LIN {X 0,Y 403.165,Z 557.03,A -85,B 0,C 180,E1 10218.684,E2 10218.684} C_VEL
LIN {X 0,Y 403.207,Z 557.03,A -85,B 0,C 180,E1 10225.722,E2 10225.722} C_VEL
LIN {X 0,Y 403.44,Z 557.03,A -85,B 0,C 180,E1 10233.237,E2 10233.237} C_VEL
LIN {X 0,Y 403.729,Z 557.03,A -85,B 0,C 180,E1 10240.276,E2 10240.276} C_VEL
LIN {X 0,Y 403.994,Z 557.03,A -85,B 0,C 180,E1 10247.007,E2 10247.007} C_VEL
LIN {X 0,Y 404.192,Z 557.03,A -85,B 0,C 180,E1 10253.549,E2 10253.549} C_VEL
LIN {X 0,Y 404.54,Z 557.03,A -85,B 0,C 180,E1 10260,E2 10260} C_VEL
LIN {X 0,Y 404.221,Z 557.03,A -85,B 0,C 180,E1 10266.452,E2 10266.452} C_VEL
LIN {X 0,Y 403.903,Z 557.03,A -85,B 0,C 180,E1 10272.997,E2 10272.997} C_VEL
LIN {X 0,Y 403.588,Z 557.03,A -85,B 0,C 180,E1 10280.305,E2 10280.305} C_VEL
LIN {X 0,Y 403.428,Z 557.03,A -85,B 0,C 180,E1 10286.765,E2 10286.765} C_VEL
LIN {X 0,Y 403.272,Z 557.03,A -85,B 0,C 180,E1 10291.708,E2 10291.708} C_VEL
LIN {X 0,Y 403.118,Z 557.03,A -85,B 0,C 180,E1 10297.934,E2 10297.934} C_VEL
LIN {X 0,Y 403.276,Z 557.65,A -85,B 0,C 180,E1 10303.8,E2 10303.8} C_VEL
LIN {X 0,Y 426.424,Z 601.688,A -85,B 0,C 180,E1 10307.749,E2 10307.749} C_VEL
LIN {X 0,Y 436.03,Z 627.386,A -85,B 0,C 180,E1 10309.651,E2 10309.651} C_VEL
LIN {X 0,Y 431.949,Z 666.261,A -85,B 0,C 180,E1 10311.298,E2 10311.298} C_VEL
LIN {X 0,Y 426.944,Z 703.511,A -85,B 0,C 180,E1 10313.718,E2 10313.718} C_VEL
LIN {X 0,Y 421.04,Z 740.02,A -85,B 0,C 180,E1 10317.052,E2 10317.052} C_VEL
LIN {X 0,Y 415.393,Z 772.458,A -85,B 0,C 180,E1 10321.118,E2 10321.118} C_VEL
LIN {X 0,Y 410.738,Z 800.362,A -85,B 0,C 180,E1 10325.811,E2 10325.811} C_VEL
LIN {X 0,Y 407.625,Z 822.502,A -85,B 0,C 180,E1 10330.852,E2 10330.852} C_VEL
LIN {X 0,Y 406.966,Z 827.151,A -85,B 0,C 180,E1 10332.15,E2 10332.15} C_VEL
LIN {X 0,Y 402.175,Z 834.199,A -85,B 0,C 180,E1 10334.327,E2 10334.327} C_VEL
LIN {X 0,Y 397.666,Z 840.297,A -85,B 0,C 180,E1 10336.6,E2 10336.6} C_VEL
LIN {X 0,Y 397.045,Z 849.258,A -85,B 0,C 180,E1 10341.227,E2 10341.227} C_VEL
LIN {X 0,Y 396.776,Z 854.259,A -85,B 0,C 180,E1 10345.623,E2 10345.623} C_VEL
LIN {X 0,Y 396.836,Z 855.967,A -85,B 0,C 180,E1 10350,E2 10350} C_VEL
LIN {X 0,Y 396.833,Z 853.357,A -85,B 0,C 180,E1 10355.474,E2 10355.474} C_VEL
LIN {X 0,Y 397.276,Z 845.463,A -85,B 0,C 180,E1 10360.986,E2 10360.986} C_VEL
LIN {X 0,Y 398.586,Z 831.788,A -85,B 0,C 180,E1 10366.553,E2 10366.553} C_VEL
LIN {X 0,Y 401.185,Z 812.548,A -85,B 0,C 180,E1 10371.881,E2 10371.881} C_VEL
LIN {X 0,Y 405.349,Z 787.469,A -85,B 0,C 180,E1 10376.93,E2 10376.93} C_VEL
LIN {X 0,Y 410.746,Z 757.402,A -85,B 0,C 180,E1 10381.419,E2 10381.419} C_VEL
LIN {X 0,Y 416.603,Z 724.967,A -85,B 0,C 180,E1 10385.02,E2 10385.02} C_VEL
LIN {X 0,Y 422.428,Z 688.774,A -85,B 0,C 180,E1 10387.958,E2 10387.958} C_VEL
LIN {X 0,Y 427.491,Z 650.452,A -85,B 0,C 180,E1 10390.101,E2 10390.101} C_VEL
LIN {X 0,Y 429.146,Z 626.905,A -85,B 0,C 180,E1 10391.084,E2 10391.084} C_VEL
LIN {X 0,Y 415.014,Z 593.65,A -85,B 0,C 180,E1 10393.806,E2 10393.806} C_VEL
LIN {X 0,Y 397.196,Z 562.149,A -85,B 0,C 180,E1 10396.941,E2 10396.941} C_VEL
LIN {X 0,Y 395.293,Z 557.03,A -85,B 0,C 180,E1 10397.449,E2 10397.449} C_VEL
LIN {X 0,Y 395.232,Z 557.03,A -85,B 0,C 180,E1 10404.929,E2 10404.929} C_VEL
LIN {X 0,Y 395.398,Z 557.03,A -85,B 0,C 180,E1 10411.729,E2 10411.729} C_VEL
LIN {X 0,Y 395.637,Z 557.03,A -85,B 0,C 180,E1 10417.501,E2 10417.501} C_VEL
LIN {X 0,Y 395.771,Z 557.03,A -85,B 0,C 180,E1 10424.468,E2 10424.468} C_VEL
LIN {X 0,Y 396.146,Z 557.03,A -85,B 0,C 180,E1 10431.206,E2 10431.206} C_VEL
LIN {X 0,Y 396.61,Z 557.03,A -85,B 0,C 180,E1 10437.812,E2 10437.812} C_VEL
LIN {X 0,Y 396.445,Z 557.03,A -85,B 0,C 180,E1 10444.38,E2 10444.38} C_VEL
LIN {X 0,Y 396.051,Z 557.03,A -85,B 0,C 180,E1 10451.018,E2 10451.018} C_VEL
LIN {X 0,Y 395.86,Z 557.03,A -85,B 0,C 180,E1 10457.815,E2 10457.815} C_VEL
LIN {X 0,Y 395.54,Z 557.03,A -85,B 0,C 180,E1 10464.899,E2 10464.899} C_VEL
LIN {X 0,Y 395.4,Z 557.03,A -85,B 0,C 180,E1 10469.851,E2 10469.851} C_VEL
LIN {X 0,Y 395.176,Z 557.03,A -85,B 0,C 180,E1 10476.43,E2 10476.43} C_VEL
LIN {X 0,Y 395.189,Z 557.03,A -85,B 0,C 180,E1 10483.595,E2 10483.595} C_VEL
LIN {X 0,Y 395.261,Z 557.03,A -85,B 0,C 180,E1 10487.074,E2 10487.074} C_VEL
LIN {X 0,Y 397.693,Z 562.671,A -85,B 0,C 180,E1 10487.578,E2 10487.578} C_VEL
LIN {X 0,Y 418.659,Z 600.152,A -85,B 0,C 180,E1 10491.241,E2 10491.241} C_VEL
LIN {X 0,Y 428.676,Z 623.291,A -85,B 0,C 180,E1 10493.314,E2 10493.314} C_VEL
LIN {X 0,Y 424.543,Z 659.037,A -85,B 0,C 180,E1 10495.067,E2 10495.067} C_VEL
LIN {X 0,Y 419.009,Z 693.568,A -85,B 0,C 180,E1 10497.653,E2 10497.653} C_VEL
LIN {X 0,Y 412.847,Z 725.198,A -85,B 0,C 180,E1 10501.077,E2 10501.077} C_VEL
LIN {X 0,Y 407.204,Z 751.222,A -85,B 0,C 180,E1 10504.979,E2 10504.979} C_VEL
LIN {X 0,Y 402.464,Z 773.712,A -85,B 0,C 180,E1 10509.636,E2 10509.636} C_VEL
LIN {X 0,Y 399.372,Z 790.725,A -85,B 0,C 180,E1 10514.61,E2 10514.61} C_VEL
LIN {X 0,Y 397.661,Z 803.103,A -85,B 0,C 180,E1 10520.134,E2 10520.134} C_VEL
LIN {X 0,Y 397.016,Z 809.778,A -85,B 0,C 180,E1 10525.625,E2 10525.625} C_VEL
LIN {X 0,Y 396.954,Z 811.42,A -85,B 0,C 180,E1 10530,E2 10530} C_VEL
LIN {X 0,Y 397.126,Z 808.803,A -85,B 0,C 180,E1 10535.469,E2 10535.469} C_VEL
LIN {X 0,Y 397.896,Z 800.917,A -85,B 0,C 180,E1 10540.967,E2 10540.967} C_VEL
LIN {X 0,Y 399.978,Z 787.154,A -85,B 0,C 180,E1 10546.493,E2 10546.493} C_VEL
LIN {X 0,Y 403.828,Z 767.438,A -85,B 0,C 180,E1 10551.73,E2 10551.73} C_VEL
LIN {X 0,Y 408.723,Z 744.251,A -85,B 0,C 180,E1 10556.097,E2 10556.097} C_VEL
LIN {X 0,Y 414.5,Z 716.892,A -85,B 0,C 180,E1 10559.846,E2 10559.846} C_VEL
LIN {X 0,Y 420.536,Z 684.985,A -85,B 0,C 180,E1 10562.993,E2 10562.993} C_VEL
LIN {X 0,Y 425.681,Z 650.957,A -85,B 0,C 180,E1 10565.307,E2 10565.307} C_VEL
LIN {X 0,Y 428.316,Z 621.671,A -85,B 0,C 180,E1 10566.708,E2 10566.708} C_VEL
LIN {X 0,Y 411.761,Z 586.807,A -85,B 0,C 180,E1 10569.882,E2 10569.882} C_VEL
LIN {X 0,Y 395.357,Z 558.405,A -85,B 0,C 180,E1 10572.754,E2 10572.754} C_VEL
LIN {X 0,Y 395.248,Z 557.03,A -85,B 0,C 180,E1 10572.937,E2 10572.937} C_VEL
LIN {X 0,Y 395.242,Z 557.03,A -85,B 0,C 180,E1 10580.008,E2 10580.008} C_VEL
LIN {X 0,Y 395.268,Z 557.03,A -85,B 0,C 180,E1 10587.574,E2 10587.574} C_VEL
LIN {X 0,Y 395.445,Z 557.03,A -85,B 0,C 180,E1 10592.651,E2 10592.651} C_VEL
LIN {X 0,Y 395.802,Z 557.03,A -85,B 0,C 180,E1 10599.864,E2 10599.864} C_VEL
LIN {X 0,Y 396.053,Z 557.03,A -85,B 0,C 180,E1 10606.741,E2 10606.741} C_VEL
LIN {X 0,Y 396.284,Z 557.03,A -85,B 0,C 180,E1 10613.419,E2 10613.419} C_VEL
LIN {X 0,Y 396.638,Z 557.03,A -85,B 0,C 180,E1 10620,E2 10620} C_VEL
LIN {X 0,Y 396.306,Z 557.03,A -85,B 0,C 180,E1 10626.637,E2 10626.637} C_VEL
LIN {X 0,Y 395.957,Z 557.03,A -85,B 0,C 180,E1 10633.263,E2 10633.263} C_VEL
LIN {X 0,Y 395.725,Z 557.03,A -85,B 0,C 180,E1 10640.141,E2 10640.141} C_VEL
LIN {X 0,Y 395.436,Z 557.03,A -85,B 0,C 180,E1 10647.35,E2 10647.35} C_VEL
LIN {X 0,Y 395.287,Z 557.03,A -85,B 0,C 180,E1 10652.579,E2 10652.579} C_VEL
LIN {X 0,Y 395.249,Z 557.03,A -85,B 0,C 180,E1 10659.993,E2 10659.993} C_VEL
LIN {X 0,Y 395.305,Z 557.034,A -85,B 0,C 180,E1 10662.665,E2 10662.665} C_VEL
LIN {X 0,Y 397.735,Z 562.702,A -85,B 0,C 180,E1 10663.162,E2 10663.162} C_VEL
LIN {X 0,Y 417.577,Z 598.711,A -85,B 0,C 180,E1 10666.649,E2 10666.649} C_VEL
LIN {X 0,Y 429.63,Z 629.235,A -85,B 0,C 180,E1 10669.068,E2 10669.068} C_VEL
LIN {X 0,Y 425.163,Z 669.268,A -85,B 0,C 180,E1 10670.836,E2 10670.836} C_VEL
LIN {X 0,Y 419.577,Z 707.742,A -85,B 0,C 180,E1 10673.459,E2 10673.459} C_VEL
LIN {X 0,Y 413.477,Z 742.914,A -85,B 0,C 180,E1 10676.845,E2 10676.845} C_VEL
LIN {X 0,Y 407.709,Z 774.237,A -85,B 0,C 180,E1 10680.937,E2 10680.937} C_VEL
LIN {X 0,Y 403.02,Z 800.884,A -85,B 0,C 180,E1 10685.592,E2 10685.592} C_VEL
LIN {X 0,Y 399.745,Z 823.015,A -85,B 0,C 180,E1 10690.796,E2 10690.796} C_VEL
LIN {X 0,Y 397.756,Z 839.4,A -85,B 0,C 180,E1 10696.238,E2 10696.238} C_VEL
LIN {X 0,Y 397.666,Z 840.297,A -85,B 0,C 180,E1 10696.6,E2 10696.6} C_VEL
LIN {X 0,Y 394.853,Z 844.248,A -85,B 0,C 180,E1 10698.366,E2 10698.366} C_VEL
LIN {X 0,Y 389.243,Z 848.814,A -85,B 0,C 180,E1 10701.079,E2 10701.079} C_VEL
LIN {X 0,Y 389.109,Z 849.256,A -85,B 0,C 180,E1 10701.397,E2 10701.397} C_VEL
LIN {X 0,Y 388.883,Z 853.803,A -85,B 0,C 180,E1 10705.534,E2 10705.534} C_VEL
LIN {X 0,Y 388.961,Z 855.525,A -85,B 0,C 180,E1 10710,E2 10710} C_VEL
LIN {X 0,Y 388.958,Z 852.896,A -85,B 0,C 180,E1 10715.585,E2 10715.585} C_VEL
LIN {X 0,Y 389.415,Z 844.941,A -85,B 0,C 180,E1 10721.21,E2 10721.21} C_VEL
LIN {X 0,Y 390.597,Z 832.802,A -85,B 0,C 180,E1 10726.322,E2 10726.322} C_VEL
LIN {X 0,Y 393.13,Z 814.175,A -85,B 0,C 180,E1 10731.758,E2 10731.758} C_VEL
LIN {X 0,Y 397.32,Z 790.516,A -85,B 0,C 180,E1 10736.792,E2 10736.792} C_VEL
LIN {X 0,Y 402.866,Z 761.455,A -85,B 0,C 180,E1 10741.398,E2 10741.398} C_VEL
LIN {X 0,Y 409.308,Z 727.729,A -85,B 0,C 180,E1 10745.337,E2 10745.337} C_VEL
LIN {X 0,Y 415.569,Z 691.107,A -85,B 0,C 180,E1 10748.421,E2 10748.421} C_VEL
LIN {X 0,Y 420.858,Z 653.779,A -85,B 0,C 180,E1 10750.596,E2 10750.596} C_VEL
LIN {X 0,Y 422.862,Z 629.874,A -85,B 0,C 180,E1 10751.636,E2 10751.636} C_VEL
LIN {X 0,Y 409.373,Z 597.325,A -85,B 0,C 180,E1 10754.401,E2 10754.401} C_VEL
LIN {X 0,Y 389.835,Z 562.756,A -85,B 0,C 180,E1 10758.002,E2 10758.002} C_VEL
LIN {X 0,Y 387.326,Z 557.03,A -85,B 0,C 180,E1 10758.636,E2 10758.636} C_VEL
LIN {X 0,Y 387.322,Z 557.03,A -85,B 0,C 180,E1 10765.175,E2 10765.175} C_VEL
LIN {X 0,Y 387.524,Z 557.03,A -85,B 0,C 180,E1 10772.043,E2 10772.043} C_VEL
LIN {X 0,Y 387.827,Z 557.03,A -85,B 0,C 180,E1 10779.546,E2 10779.546} C_VEL
LIN {X 0,Y 387.914,Z 557.03,A -85,B 0,C 180,E1 10786.457,E2 10786.457} C_VEL
LIN {X 0,Y 388.421,Z 557.03,A -85,B 0,C 180,E1 10793.285,E2 10793.285} C_VEL
LIN {X 0,Y 388.735,Z 557.03,A -85,B 0,C 180,E1 10800,E2 10800} C_VEL
LIN {X 0,Y 388.344,Z 557.03,A -85,B 0,C 180,E1 10806.716,E2 10806.716} C_VEL
LIN {X 0,Y 388.046,Z 557.03,A -85,B 0,C 180,E1 10813.537,E2 10813.537} C_VEL
LIN {X 0,Y 387.809,Z 557.03,A -85,B 0,C 180,E1 10820.569,E2 10820.569} C_VEL
LIN {X 0,Y 387.523,Z 557.03,A -85,B 0,C 180,E1 10827.956,E2 10827.956} C_VEL
LIN {X 0,Y 387.311,Z 557.03,A -85,B 0,C 180,E1 10834.822,E2 10834.822} C_VEL
LIN {X 0,Y 387.177,Z 557.03,A -85,B 0,C 180,E1 10842.012,E2 10842.012} C_VEL
LIN {X 0,Y 387.256,Z 557.03,A -85,B 0,C 180,E1 10845.866,E2 10845.866} C_VEL
LIN {X 0,Y 389.727,Z 562.663,A -85,B 0,C 180,E1 10846.407,E2 10846.407} C_VEL
LIN {X 0,Y 410.465,Z 598.787,A -85,B 0,C 180,E1 10850.187,E2 10850.187} C_VEL
LIN {X 0,Y 422.263,Z 626.321,A -85,B 0,C 180,E1 10852.752,E2 10852.752} C_VEL
LIN {X 0,Y 417.71,Z 662.884,A -85,B 0,C 180,E1 10854.634,E2 10854.634} C_VEL
LIN {X 0,Y 411.761,Z 697.232,A -85,B 0,C 180,E1 10857.345,E2 10857.345} C_VEL
LIN {X 0,Y 405.683,Z 726.809,A -85,B 0,C 180,E1 10860.67,E2 10860.67} C_VEL
LIN {X 0,Y 399.636,Z 753.308,A -85,B 0,C 180,E1 10864.772,E2 10864.772} C_VEL
LIN {X 0,Y 394.76,Z 775.372,A -85,B 0,C 180,E1 10869.514,E2 10869.514} C_VEL
LIN {X 0,Y 391.414,Z 792.87,A -85,B 0,C 180,E1 10874.938,E2 10874.938} C_VEL
LIN {X 0,Y 389.824,Z 803.564,A -85,B 0,C 180,E1 10879.934,E2 10879.934} C_VEL
LIN {X 0,Y 389.162,Z 810.223,A -85,B 0,C 180,E1 10885.537,E2 10885.537} C_VEL
LIN {X 0,Y 389.072,Z 811.863,A -85,B 0,C 180,E1 10890,E2 10890} C_VEL
LIN {X 0,Y 389.245,Z 809.254,A -85,B 0,C 180,E1 10895.58,E2 10895.58} C_VEL
LIN {X 0,Y 390.087,Z 801.385,A -85,B 0,C 180,E1 10901.19,E2 10901.19} C_VEL
LIN {X 0,Y 392.032,Z 789.292,A -85,B 0,C 180,E1 10906.26,E2 10906.26} C_VEL
LIN {X 0,Y 395.574,Z 771.558,A -85,B 0,C 180,E1 10911.322,E2 10911.322} C_VEL
LIN {X 0,Y 400.839,Z 748.189,A -85,B 0,C 180,E1 10916.046,E2 10916.046} C_VEL
LIN {X 0,Y 406.919,Z 720.875,A -85,B 0,C 180,E1 10919.998,E2 10919.998} C_VEL
LIN {X 0,Y 413.186,Z 689.835,A -85,B 0,C 180,E1 10923.225,E2 10923.225} C_VEL
LIN {X 0,Y 418.676,Z 656.143,A -85,B 0,C 180,E1 10925.681,E2 10925.681} C_VEL
LIN {X 0,Y 422.007,Z 624.706,A -85,B 0,C 180,E1 10927.261,E2 10927.261} C_VEL
LIN {X 0,Y 406.748,Z 591.728,A -85,B 0,C 180,E1 10930.396,E2 10930.396} C_VEL
LIN {X 0,Y 387.461,Z 558.663,A -85,B 0,C 180,E1 10933.931,E2 10933.931} C_VEL
LIN {X 0,Y 387.254,Z 557.03,A -85,B 0,C 180,E1 10934.205,E2 10934.205} C_VEL
LIN {X 0,Y 387.263,Z 557.03,A -85,B 0,C 180,E1 10941.436,E2 10941.436} C_VEL
LIN {X 0,Y 387.312,Z 557.03,A -85,B 0,C 180,E1 10946.823,E2 10946.823} C_VEL
LIN {X 0,Y 387.533,Z 557.03,A -85,B 0,C 180,E1 10953.972,E2 10953.972} C_VEL
LIN {X 0,Y 387.839,Z 557.03,A -85,B 0,C 180,E1 10959.538,E2 10959.538} C_VEL
LIN {X 0,Y 388.11,Z 557.03,A -85,B 0,C 180,E1 10966.465,E2 10966.465} C_VEL
LIN {X 0,Y 388.391,Z 557.03,A -85,B 0,C 180,E1 10973.285,E2 10973.285} C_VEL
LIN {X 0,Y 388.743,Z 557.03,A -85,B 0,C 180,E1 10980,E2 10980} C_VEL
LIN {X 0,Y 388.417,Z 557.03,A -85,B 0,C 180,E1 10986.715,E2 10986.715} C_VEL
LIN {X 0,Y 388.028,Z 557.03,A -85,B 0,C 180,E1 10993.539,E2 10993.539} C_VEL
LIN {X 0,Y 387.754,Z 557.03,A -85,B 0,C 180,E1 11000.573,E2 11000.573} C_VEL
LIN {X 0,Y 387.522,Z 557.03,A -85,B 0,C 180,E1 11007.957,E2 11007.957} C_VEL
LIN {X 0,Y 387.285,Z 557.03,A -85,B 0,C 180,E1 11015.9,E2 11015.9} C_VEL
LIN {X 0,Y 387.346,Z 557.03,A -85,B 0,C 180,E1 11021.455,E2 11021.455} C_VEL
LIN {X 0,Y 389.796,Z 562.725,A -85,B 0,C 180,E1 11022.006,E2 11022.006} C_VEL
LIN {X 0,Y 409.799,Z 598.084,A -85,B 0,C 180,E1 11025.683,E2 11025.683} C_VEL
LIN {X 0,Y 423.233,Z 630.882,A -85,B 0,C 180,E1 11028.452,E2 11028.452} C_VEL
LIN {X 0,Y 418.376,Z 672.307,A -85,B 0,C 180,E1 11030.371,E2 11030.371} C_VEL
LIN {X 0,Y 412.773,Z 708.514,A -85,B 0,C 180,E1 11032.921,E2 11032.921} C_VEL
LIN {X 0,Y 406.381,Z 743.419,A -85,B 0,C 180,E1 11036.354,E2 11036.354} C_VEL
LIN {X 0,Y 400.543,Z 773.668,A -85,B 0,C 180,E1 11040.382,E2 11040.382} C_VEL
LIN {X 0,Y 395.53,Z 800.233,A -85,B 0,C 180,E1 11045.098,E2 11045.098} C_VEL
LIN {X 0,Y 392.058,Z 822.04,A -85,B 0,C 180,E1 11050.321,E2 11050.321} C_VEL
LIN {X 0,Y 389.986,Z 838.416,A -85,B 0,C 180,E1 11055.79,E2 11055.79} C_VEL
LIN {X 0,Y 389.109,Z 849.256,A -85,B 0,C 180,E1 11061.397,E2 11061.397} C_VEL
LIN {X 0,Y 387.723,Z 850.914,A -85,B 0,C 180,E1 11062.645,E2 11062.645} C_VEL
LIN {X 0,Y 380.923,Z 853.959,A -85,B 0,C 180,E1 11066.339,E2 11066.339} C_VEL
LIN {X 0,Y 380.915,Z 853.897,A -85,B 0,C 180,E1 11066.421,E2 11066.421} C_VEL
LIN {X 0,Y 381.072,Z 855.082,A -85,B 0,C 180,E1 11070,E2 11070} C_VEL
LIN {X 0,Y 380.996,Z 853.345,A -85,B 0,C 180,E1 11074.559,E2 11074.559} C_VEL
LIN {X 0,Y 381.423,Z 846.471,A -85,B 0,C 180,E1 11080.29,E2 11080.29} C_VEL
LIN {X 0,Y 382.457,Z 835.419,A -85,B 0,C 180,E1 11085.499,E2 11085.499} C_VEL
LIN {X 0,Y 385.001,Z 817.102,A -85,B 0,C 180,E1 11091.31,E2 11091.31} C_VEL
LIN {X 0,Y 389.227,Z 793.518,A -85,B 0,C 180,E1 11096.653,E2 11096.653} C_VEL
LIN {X 0,Y 394.728,Z 766.59,A -85,B 0,C 180,E1 11101.186,E2 11101.186} C_VEL
LIN {X 0,Y 401.037,Z 735.014,A -85,B 0,C 180,E1 11105.172,E2 11105.172} C_VEL
LIN {X 0,Y 407.747,Z 699.7,A -85,B 0,C 180,E1 11108.414,E2 11108.414} C_VEL
LIN {X 0,Y 413.272,Z 664.179,A -85,B 0,C 180,E1 11110.736,E2 11110.736} C_VEL
LIN {X 0,Y 416.352,Z 632.035,A -85,B 0,C 180,E1 11112.272,E2 11112.272} C_VEL
LIN {X 0,Y 403.663,Z 600.934,A -85,B 0,C 180,E1 11115.029,E2 11115.029} C_VEL
LIN {X 0,Y 385.101,Z 568.091,A -85,B 0,C 180,E1 11118.578,E2 11118.578} C_VEL
LIN {X 0,Y 379.519,Z 558.27,A -85,B 0,C 180,E1 11119.75,E2 11119.75} C_VEL
LIN {X 0,Y 379.451,Z 557.03,A -85,B 0,C 180,E1 11119.859,E2 11119.859} C_VEL
LIN {X 0,Y 379.436,Z 557.03,A -85,B 0,C 180,E1 11126.926,E2 11126.926} C_VEL
LIN {X 0,Y 379.643,Z 557.03,A -85,B 0,C 180,E1 11133.981,E2 11133.981} C_VEL
LIN {X 0,Y 379.912,Z 557.03,A -85,B 0,C 180,E1 11141.409,E2 11141.409} C_VEL
LIN {X 0,Y 380.062,Z 557.03,A -85,B 0,C 180,E1 11148.511,E2 11148.511} C_VEL
LIN {X 0,Y 380.523,Z 557.03,A -85,B 0,C 180,E1 11155.436,E2 11155.436} C_VEL
LIN {X 0,Y 380.834,Z 557.03,A -85,B 0,C 180,E1 11160,E2 11160} C_VEL
LIN {X 0,Y 380.433,Z 557.03,A -85,B 0,C 180,E1 11166.856,E2 11166.856} C_VEL
LIN {X 0,Y 380.103,Z 557.03,A -85,B 0,C 180,E1 11173.826,E2 11173.826} C_VEL
LIN {X 0,Y 379.831,Z 557.03,A -85,B 0,C 180,E1 11181.021,E2 11181.021} C_VEL
LIN {X 0,Y 379.527,Z 557.03,A -85,B 0,C 180,E1 11188.639,E2 11188.639} C_VEL
LIN {X 0,Y 379.375,Z 557.03,A -85,B 0,C 180,E1 11193.965,E2 11193.965} C_VEL
LIN {X 0,Y 379.212,Z 557.03,A -85,B 0,C 180,E1 11200.659,E2 11200.659} C_VEL
LIN {X 0,Y 379.31,Z 557.559,A -85,B 0,C 180,E1 11204.628,E2 11204.628} C_VEL
LIN {X 0,Y 381.988,Z 562.965,A -85,B 0,C 180,E1 11205.205,E2 11205.205} C_VEL
LIN {X 0,Y 402.845,Z 598.459,A -85,B 0,C 180,E1 11209.186,E2 11209.186} C_VEL
LIN {X 0,Y 415.904,Z 629.213,A -85,B 0,C 180,E1 11212.167,E2 11212.167} C_VEL
LIN {X 0,Y 410.844,Z 666.49,A -85,B 0,C 180,E1 11214.186,E2 11214.186} C_VEL
LIN {X 0,Y 404.765,Z 699.746,A -85,B 0,C 180,E1 11216.927,E2 11216.927} C_VEL
LIN {X 0,Y 398.286,Z 729.434,A -85,B 0,C 180,E1 11220.384,E2 11220.384} C_VEL
LIN {X 0,Y 392.086,Z 755.387,A -85,B 0,C 180,E1 11224.558,E2 11224.558} C_VEL
LIN {X 0,Y 387.036,Z 776.93,A -85,B 0,C 180,E1 11229.385,E2 11229.385} C_VEL
LIN {X 0,Y 383.753,Z 793.018,A -85,B 0,C 180,E1 11234.498,E2 11234.498} C_VEL
LIN {X 0,Y 382.004,Z 804.022,A -85,B 0,C 180,E1 11239.726,E2 11239.726} C_VEL
LIN {X 0,Y 381.28,Z 810.669,A -85,B 0,C 180,E1 11245.444,E2 11245.444} C_VEL
LIN {X 0,Y 381.184,Z 812.305,A -85,B 0,C 180,E1 11250,E2 11250} C_VEL
LIN {X 0,Y 381.389,Z 809.703,A -85,B 0,C 180,E1 11255.695,E2 11255.695} C_VEL
LIN {X 0,Y 382.278,Z 801.851,A -85,B 0,C 180,E1 11261.421,E2 11261.421} C_VEL
LIN {X 0,Y 384.361,Z 789.777,A -85,B 0,C 180,E1 11266.594,E2 11266.594} C_VEL
LIN {X 0,Y 388.17,Z 772.065,A -85,B 0,C 180,E1 11271.749,E2 11271.749} C_VEL
LIN {X 0,Y 393.691,Z 748.737,A -85,B 0,C 180,E1 11276.556,E2 11276.556} C_VEL
LIN {X 0,Y 400.327,Z 720.368,A -85,B 0,C 180,E1 11280.702,E2 11280.702} C_VEL
LIN {X 0,Y 406.818,Z 689.418,A -85,B 0,C 180,E1 11283.935,E2 11283.935} C_VEL
LIN {X 0,Y 412.439,Z 656.42,A -85,B 0,C 180,E1 11286.352,E2 11286.352} C_VEL
LIN {X 0,Y 415.534,Z 627.287,A -85,B 0,C 180,E1 11287.877,E2 11287.877} C_VEL
LIN {X 0,Y 400.346,Z 593.876,A -85,B 0,C 180,E1 11291.19,E2 11291.19} C_VEL
LIN {X 0,Y 381.136,Z 562.063,A -85,B 0,C 180,E1 11294.847,E2 11294.847} C_VEL
LIN {X 0,Y 379.333,Z 557.03,A -85,B 0,C 180,E1 11295.304,E2 11295.304} C_VEL
LIN {X 0,Y 379.252,Z 557.03,A -85,B 0,C 180,E1 11300.305,E2 11300.305} C_VEL
LIN {X 0,Y 379.427,Z 557.03,A -85,B 0,C 180,E1 11306.926,E2 11306.926} C_VEL
LIN {X 0,Y 379.649,Z 557.03,A -85,B 0,C 180,E1 11313.983,E2 11313.983} C_VEL
LIN {X 0,Y 380.001,Z 557.03,A -85,B 0,C 180,E1 11321.415,E2 11321.415} C_VEL
LIN {X 0,Y 380.271,Z 557.03,A -85,B 0,C 180,E1 11328.518,E2 11328.518} C_VEL
LIN {X 0,Y 380.618,Z 557.03,A -85,B 0,C 180,E1 11335.438,E2 11335.438} C_VEL
LIN {X 0,Y 380.795,Z 557.03,A -85,B 0,C 180,E1 11342.279,E2 11342.279} C_VEL
LIN {X 0,Y 380.311,Z 557.03,A -85,B 0,C 180,E1 11349.163,E2 11349.163} C_VEL
LIN {X 0,Y 379.967,Z 557.03,A -85,B 0,C 180,E1 11356.196,E2 11356.196} C_VEL
LIN {X 0,Y 379.716,Z 557.03,A -85,B 0,C 180,E1 11363.498,E2 11363.498} C_VEL
LIN {X 0,Y 379.415,Z 557.03,A -85,B 0,C 180,E1 11371.247,E2 11371.247} C_VEL
LIN {X 0,Y 379.283,Z 557.03,A -85,B 0,C 180,E1 11377.025,E2 11377.025} C_VEL
LIN {X 0,Y 379.431,Z 557.03,A -85,B 0,C 180,E1 11380.203,E2 11380.203} C_VEL
LIN {X 0,Y 381.795,Z 562.637,A -85,B 0,C 180,E1 11380.761,E2 11380.761} C_VEL
LIN {X 0,Y 401.064,Z 595.734,A -85,B 0,C 180,E1 11384.483,E2 11384.483} C_VEL
LIN {X 0,Y 414.31,Z 626.287,A -85,B 0,C 180,E1 11387.245,E2 11387.245} C_VEL
LIN {X 0,Y 416.724,Z 634.752,A -85,B 0,C 180,E1 11387.912,E2 11387.912} C_VEL
LIN {X 0,Y 411.832,Z 673.531,A -85,B 0,C 180,E1 11389.785,E2 11389.785} C_VEL
LIN {X 0,Y 405.961,Z 709.471,A -85,B 0,C 180,E1 11392.377,E2 11392.377} C_VEL
LIN {X 0,Y 399.361,Z 743.852,A -85,B 0,C 180,E1 11395.836,E2 11395.836} C_VEL
LIN {X 0,Y 393.176,Z 774.118,A -85,B 0,C 180,E1 11399.96,E2 11399.96} C_VEL
LIN {X 0,Y 387.84,Z 801.02,A -85,B 0,C 180,E1 11404.879,E2 11404.879} C_VEL
LIN {X 0,Y 384.158,Z 822.955,A -85,B 0,C 180,E1 11410.337,E2 11410.337} C_VEL
LIN {X 0,Y 381.967,Z 839.667,A -85,B 0,C 180,E1 11416.242,E2 11416.242} C_VEL
LIN {X 0,Y 381.172,Z 849.92,A -85,B 0,C 180,E1 11422.009,E2 11422.009} C_VEL
LIN {X 0,Y 380.915,Z 853.897,A -85,B 0,C 180,E1 11426.421,E2 11426.421} C_VEL
LIN {X 0,Y 378.401,Z 854.68,A -85,B 0,C 180,E1 11428.361,E2 11428.361} C_VEL
LIN {X 0,Y 373.165,Z 854.446,A -85,B 0,C 180,E1 11431.291,E2 11431.291} C_VEL
LIN {X 0,Y 373.082,Z 854.32,A -85,B 0,C 180,E1 11431.63,E2 11431.63} C_VEL
LIN {X 0,Y 373.224,Z 850.761,A -85,B 0,C 180,E1 11436.991,E2 11436.991} C_VEL
LIN {X 0,Y 373.918,Z 841.866,A -85,B 0,C 180,E1 11442.741,E2 11442.741} C_VEL
LIN {X 0,Y 375.548,Z 828.32,A -85,B 0,C 180,E1 11448.207,E2 11448.207} C_VEL
LIN {X 0,Y 378.856,Z 808.257,A -85,B 0,C 180,E1 11453.869,E2 11453.869} C_VEL
LIN {X 0,Y 383.938,Z 783.144,A -85,B 0,C 180,E1 11459.036,E2 11459.036} C_VEL
LIN {X 0,Y 390.335,Z 753.565,A -85,B 0,C 180,E1 11463.548,E2 11463.548} C_VEL
LIN {X 0,Y 397.159,Z 720.956,A -85,B 0,C 180,E1 11467.224,E2 11467.224} C_VEL
LIN {X 0,Y 403.984,Z 683.397,A -85,B 0,C 180,E1 11470.278,E2 11470.278} C_VEL
LIN {X 0,Y 409.731,Z 643.204,A -85,B 0,C 180,E1 11472.452,E2 11472.452} C_VEL
LIN {X 0,Y 409.991,Z 634.595,A -85,B 0,C 180,E1 11472.881,E2 11472.881} C_VEL
LIN {X 0,Y 398.341,Z 605.249,A -85,B 0,C 180,E1 11475.608,E2 11475.608} C_VEL
LIN {X 0,Y 380.757,Z 573.73,A -85,B 0,C 180,E1 11479.105,E2 11479.105} C_VEL
LIN {X 0,Y 371.492,Z 558.119,A -85,B 0,C 180,E1 11481.121,E2 11481.121} C_VEL
LIN {X 0,Y 371.41,Z 557.03,A -85,B 0,C 180,E1 11481.204,E2 11481.204} C_VEL
LIN {X 0,Y 371.509,Z 557.03,A -85,B 0,C 180,E1 11488.853,E2 11488.853} C_VEL
LIN {X 0,Y 371.743,Z 557.03,A -85,B 0,C 180,E1 11495.967,E2 11495.967} C_VEL
LIN {X 0,Y 371.95,Z 557.03,A -85,B 0,C 180,E1 11500.996,E2 11500.996} C_VEL
LIN {X 0,Y 372.122,Z 557.03,A -85,B 0,C 180,E1 11508.263,E2 11508.263} C_VEL
LIN {X 0,Y 372.613,Z 557.03,A -85,B 0,C 180,E1 11515.339,E2 11515.339} C_VEL
LIN {X 0,Y 372.932,Z 557.03,A -85,B 0,C 180,E1 11520,E2 11520} C_VEL
LIN {X 0,Y 372.507,Z 557.03,A -85,B 0,C 180,E1 11527.003,E2 11527.003} C_VEL
LIN {X 0,Y 372.16,Z 557.03,A -85,B 0,C 180,E1 11534.127,E2 11534.127} C_VEL
LIN {X 0,Y 371.857,Z 557.03,A -85,B 0,C 180,E1 11541.494,E2 11541.494} C_VEL
LIN {X 0,Y 371.642,Z 557.03,A -85,B 0,C 180,E1 11546.622,E2 11546.622} C_VEL
LIN {X 0,Y 371.489,Z 557.03,A -85,B 0,C 180,E1 11551.991,E2 11551.991} C_VEL
LIN {X 0,Y 371.271,Z 557.03,A -85,B 0,C 180,E1 11559.21,E2 11559.21} C_VEL
LIN {X 0,Y 371.304,Z 557.03,A -85,B 0,C 180,E1 11563.217,E2 11563.217} C_VEL
LIN {X 0,Y 373.599,Z 562.571,A -85,B 0,C 180,E1 11563.793,E2 11563.793} C_VEL
LIN {X 0,Y 392.02,Z 592.498,A -85,B 0,C 180,E1 11567.498,E2 11567.498} C_VEL
LIN {X 0,Y 406.924,Z 624.183,A -85,B 0,C 180,E1 11570.818,E2 11570.818} C_VEL
LIN {X 0,Y 409.369,Z 633.438,A -85,B 0,C 180,E1 11571.63,E2 11571.63} C_VEL
LIN {X 0,Y 404.25,Z 668.689,A -85,B 0,C 180,E1 11573.634,E2 11573.634} C_VEL
LIN {X 0,Y 397.989,Z 701.283,A -85,B 0,C 180,E1 11576.396,E2 11576.396} C_VEL
LIN {X 0,Y 391.424,Z 730.008,A -85,B 0,C 180,E1 11579.811,E2 11579.811} C_VEL
LIN {X 0,Y 384.891,Z 755.918,A -85,B 0,C 180,E1 11584.047,E2 11584.047} C_VEL
LIN {X 0,Y 379.568,Z 777.42,A -85,B 0,C 180,E1 11588.961,E2 11588.961} C_VEL
LIN {X 0,Y 376.065,Z 793.516,A -85,B 0,C 180,E1 11594.184,E2 11594.184} C_VEL
LIN {X 0,Y 374.185,Z 804.478,A -85,B 0,C 180,E1 11599.509,E2 11599.509} C_VEL
LIN {X 0,Y 373.399,Z 811.115,A -85,B 0,C 180,E1 11605.348,E2 11605.348} C_VEL
LIN {X 0,Y 373.303,Z 812.748,A -85,B 0,C 180,E1 11610,E2 11610} C_VEL
LIN {X 0,Y 373.53,Z 810.154,A -85,B 0,C 180,E1 11615.812,E2 11615.812} C_VEL
LIN {X 0,Y 374.49,Z 802.313,A -85,B 0,C 180,E1 11621.662,E2 11621.662} C_VEL
LIN {X 0,Y 376.708,Z 790.259,A -85,B 0,C 180,E1 11626.941,E2 11626.941} C_VEL
LIN {X 0,Y 380.762,Z 772.568,A -85,B 0,C 180,E1 11632.194,E2 11632.194} C_VEL
LIN {X 0,Y 386.575,Z 749.274,A -85,B 0,C 180,E1 11637.084,E2 11637.084} C_VEL
LIN {X 0,Y 393.526,Z 720.974,A -85,B 0,C 180,E1 11641.291,E2 11641.291} C_VEL
LIN {X 0,Y 400.303,Z 690.115,A -85,B 0,C 180,E1 11644.564,E2 11644.564} C_VEL
LIN {X 0,Y 406.086,Z 657.703,A -85,B 0,C 180,E1 11646.982,E2 11646.982} C_VEL
LIN {X 0,Y 409.199,Z 630.078,A -85,B 0,C 180,E1 11648.49,E2 11648.49} C_VEL
LIN {X 0,Y 394.226,Z 596.613,A -85,B 0,C 180,E1 11651.962,E2 11651.962} C_VEL
LIN {X 0,Y 374.022,Z 562.946,A -85,B 0,C 180,E1 11656.012,E2 11656.012} C_VEL
LIN {X 0,Y 371.47,Z 558.414,A -85,B 0,C 180,E1 11656.58,E2 11656.58} C_VEL
LIN {X 0,Y 371.358,Z 557.03,A -85,B 0,C 180,E1 11656.708,E2 11656.708} C_VEL
LIN {X 0,Y 371.29,Z 557.03,A -85,B 0,C 180,E1 11662.293,E2 11662.293} C_VEL
LIN {X 0,Y 371.504,Z 557.03,A -85,B 0,C 180,E1 11668.853,E2 11668.853} C_VEL
LIN {X 0,Y 371.739,Z 557.03,A -85,B 0,C 180,E1 11675.968,E2 11675.968} C_VEL
LIN {X 0,Y 372.184,Z 557.03,A -85,B 0,C 180,E1 11683.457,E2 11683.457} C_VEL
LIN {X 0,Y 372.421,Z 557.03,A -85,B 0,C 180,E1 11690.642,E2 11690.642} C_VEL
LIN {X 0,Y 372.836,Z 557.03,A -85,B 0,C 180,E1 11697.673,E2 11697.673} C_VEL
LIN {X 0,Y 372.879,Z 557.03,A -85,B 0,C 180,E1 11702.327,E2 11702.327} C_VEL
LIN {X 0,Y 372.372,Z 557.03,A -85,B 0,C 180,E1 11709.36,E2 11709.36} C_VEL
LIN {X 0,Y 372.055,Z 557.03,A -85,B 0,C 180,E1 11716.55,E2 11716.55} C_VEL
LIN {X 0,Y 371.738,Z 557.03,A -85,B 0,C 180,E1 11724.033,E2 11724.033} C_VEL
LIN {X 0,Y 371.486,Z 557.03,A -85,B 0,C 180,E1 11731.992,E2 11731.992} C_VEL
LIN {X 0,Y 371.394,Z 557.03,A -85,B 0,C 180,E1 11738.845,E2 11738.845} C_VEL
LIN {X 0,Y 373.811,Z 562.605,A -85,B 0,C 180,E1 11739.436,E2 11739.436} C_VEL
LIN {X 0,Y 393.198,Z 595.069,A -85,B 0,C 180,E1 11743.379,E2 11743.379} C_VEL
LIN {X 0,Y 406.902,Z 625.475,A -85,B 0,C 180,E1 11746.32,E2 11746.32} C_VEL
LIN {X 0,Y 410.295,Z 637.739,A -85,B 0,C 180,E1 11747.329,E2 11747.329} C_VEL
LIN {X 0,Y 405.186,Z 675.863,A -85,B 0,C 180,E1 11749.251,E2 11749.251} C_VEL
LIN {X 0,Y 399.081,Z 711.121,A -85,B 0,C 180,E1 11751.877,E2 11751.877} C_VEL
LIN {X 0,Y 392.367,Z 744.375,A -85,B 0,C 180,E1 11755.309,E2 11755.309} C_VEL
LIN {X 0,Y 386.069,Z 773.5,A -85,B 0,C 180,E1 11759.348,E2 11759.348} C_VEL
LIN {X 0,Y 380.698,Z 799.054,A -85,B 0,C 180,E1 11764.058,E2 11764.058} C_VEL
LIN {X 0,Y 376.759,Z 820.663,A -85,B 0,C 180,E1 11769.413,E2 11769.413} C_VEL
LIN {X 0,Y 374.504,Z 836.32,A -85,B 0,C 180,E1 11774.765,E2 11774.765} C_VEL
LIN {X 0,Y 373.428,Z 847.778,A -85,B 0,C 180,E1 11780.667,E2 11780.667} C_VEL
LIN {X 0,Y 373.033,Z 853.486,A -85,B 0,C 180,E1 11786.424,E2 11786.424} C_VEL
LIN {X 0,Y 373.082,Z 854.32,A -85,B 0,C 180,E1 11791.63,E2 11791.63} C_VEL
LIN {X 0,Y 370.563,Z 853.472,A -85,B 0,C 180,E1 11793.61,E2 11793.61} C_VEL
LIN {X 0,Y 365.361,Z 850.91,A -85,B 0,C 180,E1 11796.579,E2 11796.579} C_VEL
LIN {X 0,Y 365.315,Z 850.519,A -85,B 0,C 180,E1 11796.921,E2 11796.921} C_VEL
LIN {X 0,Y 366.073,Z 841.58,A -85,B 0,C 180,E1 11802.918,E2 11802.918} C_VEL
LIN {X 0,Y 367.932,Z 827.074,A -85,B 0,C 180,E1 11808.845,E2 11808.845} C_VEL
LIN {X 0,Y 371.369,Z 807.71,A -85,B 0,C 180,E1 11814.381,E2 11814.381} C_VEL
LIN {X 0,Y 376.691,Z 782.944,A -85,B 0,C 180,E1 11819.574,E2 11819.574} C_VEL
LIN {X 0,Y 383.397,Z 753.582,A -85,B 0,C 180,E1 11824.137,E2 11824.137} C_VEL
LIN {X 0,Y 390.39,Z 721.754,A -85,B 0,C 180,E1 11827.798,E2 11827.798} C_VEL
LIN {X 0,Y 397.137,Z 686.433,A -85,B 0,C 180,E1 11830.759,E2 11830.759} C_VEL
LIN {X 0,Y 403.106,Z 647.847,A -85,B 0,C 180,E1 11832.964,E2 11832.964} C_VEL
LIN {X 0,Y 403.708,Z 637.185,A -85,B 0,C 180,E1 11833.5,E2 11833.5} C_VEL
LIN {X 0,Y 392.192,Z 607.731,A -85,B 0,C 180,E1 11836.368,E2 11836.368} C_VEL
LIN {X 0,Y 373.793,Z 574.786,A -85,B 0,C 180,E1 11840.223,E2 11840.223} C_VEL
LIN {X 0,Y 363.494,Z 558.064,A -85,B 0,C 180,E1 11842.586,E2 11842.586} C_VEL
LIN {X 0,Y 363.424,Z 557.03,A -85,B 0,C 180,E1 11842.746,E2 11842.746} C_VEL
LIN {X 0,Y 363.615,Z 557.03,A -85,B 0,C 180,E1 11850.024,E2 11850.024} C_VEL
LIN {X 0,Y 363.878,Z 557.03,A -85,B 0,C 180,E1 11858.009,E2 11858.009} C_VEL
LIN {X 0,Y 364.108,Z 557.03,A -85,B 0,C 180,E1 11865.553,E2 11865.553} C_VEL
LIN {X 0,Y 364.662,Z 557.03,A -85,B 0,C 180,E1 11872.845,E2 11872.845} C_VEL
LIN {X 0,Y 365.03,Z 557.03,A -85,B 0,C 180,E1 11880,E2 11880} C_VEL
LIN {X 0,Y 364.585,Z 557.03,A -85,B 0,C 180,E1 11887.156,E2 11887.156} C_VEL
LIN {X 0,Y 364.216,Z 557.03,A -85,B 0,C 180,E1 11894.442,E2 11894.442} C_VEL
LIN {X 0,Y 363.876,Z 557.03,A -85,B 0,C 180,E1 11901.99,E2 11901.99} C_VEL
LIN {X 0,Y 363.614,Z 557.03,A -85,B 0,C 180,E1 11909.975,E2 11909.975} C_VEL
LIN {X 0,Y 363.373,Z 557.03,A -85,B 0,C 180,E1 11917.658,E2 11917.658} C_VEL
LIN {X 0,Y 363.406,Z 557.521,A -85,B 0,C 180,E1 11921.801,E2 11921.801} C_VEL
LIN {X 0,Y 365.947,Z 562.812,A -85,B 0,C 180,E1 11922.431,E2 11922.431} C_VEL
LIN {X 0,Y 385.714,Z 594.655,A -85,B 0,C 180,E1 11926.625,E2 11926.625} C_VEL
LIN {X 0,Y 400.188,Z 625.792,A -85,B 0,C 180,E1 11930.043,E2 11930.043} C_VEL
LIN {X 0,Y 403.16,Z 635.392,A -85,B 0,C 180,E1 11930.984,E2 11930.984} C_VEL
LIN {X 0,Y 397.688,Z 671.012,A -85,B 0,C 180,E1 11933.076,E2 11933.076} C_VEL
LIN {X 0,Y 390.819,Z 704.673,A -85,B 0,C 180,E1 11936.033,E2 11936.033} C_VEL
LIN {X 0,Y 383.311,Z 735.398,A -85,B 0,C 180,E1 11939.916,E2 11939.916} C_VEL
LIN {X 0,Y 376.535,Z 760.836,A -85,B 0,C 180,E1 11944.422,E2 11944.422} C_VEL
LIN {X 0,Y 371.327,Z 780.87,A -85,B 0,C 180,E1 11949.365,E2 11949.365} C_VEL
LIN {X 0,Y 367.858,Z 796.854,A -85,B 0,C 180,E1 11955.032,E2 11955.032} C_VEL
LIN {X 0,Y 366.181,Z 806.738,A -85,B 0,C 180,E1 11960.48,E2 11960.48} C_VEL
LIN {X 0,Y 365.52,Z 811.56,A -85,B 0,C 180,E1 11965.248,E2 11965.248} C_VEL
LIN {X 0,Y 365.415,Z 813.19,A -85,B 0,C 180,E1 11970,E2 11970} C_VEL
LIN {X 0,Y 365.535,Z 811.492,A -85,B 0,C 180,E1 11974.751,E2 11974.751} C_VEL
LIN {X 0,Y 366.403,Z 804.789,A -85,B 0,C 180,E1 11980.716,E2 11980.716} C_VEL
LIN {X 0,Y 368.733,Z 792.387,A -85,B 0,C 180,E1 11986.703,E2 11986.703} C_VEL
LIN {X 0,Y 373.076,Z 774.218,A -85,B 0,C 180,E1 11992.362,E2 11992.362} C_VEL
LIN {X 0,Y 379.069,Z 751.346,A -85,B 0,C 180,E1 11997.343,E2 11997.343} C_VEL
LIN {X 0,Y 386.264,Z 723.812,A -85,B 0,C 180,E1 12001.618,E2 12001.618} C_VEL
LIN {X 0,Y 393.532,Z 692.309,A -85,B 0,C 180,E1 12005.078,E2 12005.078} C_VEL
LIN {X 0,Y 399.656,Z 659.701,A -85,B 0,C 180,E1 12007.587,E2 12007.587} C_VEL
LIN {X 0,Y 402.952,Z 633.102,A -85,B 0,C 180,E1 12009.086,E2 12009.086} C_VEL
LIN {X 0,Y 388.682,Z 600.276,A -85,B 0,C 180,E1 12012.626,E2 12012.626} C_VEL
LIN {X 0,Y 369.853,Z 568.768,A -85,B 0,C 180,E1 12016.584,E2 12016.584} C_VEL
LIN {X 0,Y 363.577,Z 558.452,A -85,B 0,C 180,E1 12018.023,E2 12018.023} C_VEL
LIN {X 0,Y 363.434,Z 557.03,A -85,B 0,C 180,E1 12018.203,E2 12018.203} C_VEL
LIN {X 0,Y 363.385,Z 557.03,A -85,B 0,C 180,E1 12024.32,E2 12024.32} C_VEL
LIN {X 0,Y 363.662,Z 557.03,A -85,B 0,C 180,E1 12030.962,E2 12030.962} C_VEL
LIN {X 0,Y 363.882,Z 557.03,A -85,B 0,C 180,E1 12038.01,E2 12038.01} C_VEL
LIN {X 0,Y 364.305,Z 557.03,A -85,B 0,C 180,E1 12045.562,E2 12045.562} C_VEL
LIN {X 0,Y 364.639,Z 557.03,A -85,B 0,C 180,E1 12052.845,E2 12052.845} C_VEL
LIN {X 0,Y 365.038,Z 557.03,A -85,B 0,C 180,E1 12060,E2 12060} C_VEL
LIN {X 0,Y 364.665,Z 557.03,A -85,B 0,C 180,E1 12067.155,E2 12067.155} C_VEL
LIN {X 0,Y 364.186,Z 557.03,A -85,B 0,C 180,E1 12074.444,E2 12074.444} C_VEL
LIN {X 0,Y 363.85,Z 557.03,A -85,B 0,C 180,E1 12081.993,E2 12081.993} C_VEL
LIN {X 0,Y 363.611,Z 557.03,A -85,B 0,C 180,E1 12089.976,E2 12089.976} C_VEL
LIN {X 0,Y 363.456,Z 557.742,A -85,B 0,C 180,E1 12097.419,E2 12097.419} C_VEL
LIN {X 0,Y 366.283,Z 563.05,A -85,B 0,C 180,E1 12098.114,E2 12098.114} C_VEL
LIN {X 0,Y 386.389,Z 596.357,A -85,B 0,C 180,E1 12102.428,E2 12102.428} C_VEL
LIN {X 0,Y 400.282,Z 626.878,A -85,B 0,C 180,E1 12105.553,E2 12105.553} C_VEL
LIN {X 0,Y 403.952,Z 640.514,A -85,B 0,C 180,E1 12106.72,E2 12106.72} C_VEL
LIN {X 0,Y 398.374,Z 679.291,A -85,B 0,C 180,E1 12108.765,E2 12108.765} C_VEL
LIN {X 0,Y 391.327,Z 717.197,A -85,B 0,C 180,E1 12111.754,E2 12111.754} C_VEL
LIN {X 0,Y 383.857,Z 751.557,A -85,B 0,C 180,E1 12115.596,E2 12115.596} C_VEL
LIN {X 0,Y 377.01,Z 781.692,A -85,B 0,C 180,E1 12120.208,E2 12120.208} C_VEL
LIN {X 0,Y 371.594,Z 806.443,A -85,B 0,C 180,E1 12125.315,E2 12125.315} C_VEL
LIN {X 0,Y 367.987,Z 826.987,A -85,B 0,C 180,E1 12131.13,E2 12131.13} C_VEL
LIN {X 0,Y 366.011,Z 841.63,A -85,B 0,C 180,E1 12137.107,E2 12137.107} C_VEL
LIN {X 0,Y 365.345,Z 850.297,A -85,B 0,C 180,E1 12142.859,E2 12142.859} C_VEL
LIN {X 0,Y 365.207,Z 853.735,A -85,B 0,C 180,E1 12147.624,E2 12147.624} C_VEL
LIN {X 0,Y 365.228,Z 853.737,A -85,B 0,C 180,E1 12152.376,E2 12152.376} C_VEL
LIN {X 0,Y 365.315,Z 850.519,A -85,B 0,C 180,E1 12156.921,E2 12156.921} C_VEL
LIN {X 0,Y 363.014,Z 848.188,A -85,B 0,C 180,E1 12158.92,E2 12158.92} C_VEL
LIN {X 0,Y 358.04,Z 843.533,A -85,B 0,C 180,E1 12161.894,E2 12161.894} C_VEL
LIN {X 0,Y 358.014,Z 842.92,A -85,B 0,C 180,E1 12162.234,E2 12162.234} C_VEL
LIN {X 0,Y 359.948,Z 828.518,A -85,B 0,C 180,E1 12168.599,E2 12168.599} C_VEL
LIN {X 0,Y 363.665,Z 808.435,A -85,B 0,C 180,E1 12174.604,E2 12174.604} C_VEL
LIN {X 0,Y 369.14,Z 784.185,A -85,B 0,C 180,E1 12179.872,E2 12179.872} C_VEL
LIN {X 0,Y 376.143,Z 755.011,A -85,B 0,C 180,E1 12184.559,E2 12184.559} C_VEL
LIN {X 0,Y 383.576,Z 722.895,A -85,B 0,C 180,E1 12188.36,E2 12188.36} C_VEL
LIN {X 0,Y 390.683,Z 687.547,A -85,B 0,C 180,E1 12191.395,E2 12191.395} C_VEL
LIN {X 0,Y 396.775,Z 650.224,A -85,B 0,C 180,E1 12193.59,E2 12193.59} C_VEL
LIN {X 0,Y 397.348,Z 639.282,A -85,B 0,C 180,E1 12194.182,E2 12194.182} C_VEL
LIN {X 0,Y 386.318,Z 610.895,A -85,B 0,C 180,E1 12197.085,E2 12197.085} C_VEL
LIN {X 0,Y 369.431,Z 580.236,A -85,B 0,C 180,E1 12200.813,E2 12200.813} C_VEL
LIN {X 0,Y 357.44,Z 562.257,A -85,B 0,C 180,E1 12203.631,E2 12203.631} C_VEL
LIN {X 0,Y 355.501,Z 557.03,A -85,B 0,C 180,E1 12204.295,E2 12204.295} C_VEL
LIN {X 0,Y 355.738,Z 557.03,A -85,B 0,C 180,E1 12212.086,E2 12212.086} C_VEL
LIN {X 0,Y 356.057,Z 557.03,A -85,B 0,C 180,E1 12220.113,E2 12220.113} C_VEL
LIN {X 0,Y 356.281,Z 557.03,A -85,B 0,C 180,E1 12227.8,E2 12227.8} C_VEL
LIN {X 0,Y 356.826,Z 557.03,A -85,B 0,C 180,E1 12235.132,E2 12235.132} C_VEL
LIN {X 0,Y 357.142,Z 557.03,A -85,B 0,C 180,E1 12240,E2 12240} C_VEL
LIN {X 0,Y 356.654,Z 557.03,A -85,B 0,C 180,E1 12247.316,E2 12247.316} C_VEL
LIN {X 0,Y 356.272,Z 557.03,A -85,B 0,C 180,E1 12254.771,E2 12254.771} C_VEL
LIN {X 0,Y 355.924,Z 557.03,A -85,B 0,C 180,E1 12262.508,E2 12262.508} C_VEL
LIN {X 0,Y 355.739,Z 557.03,A -85,B 0,C 180,E1 12267.913,E2 12267.913} C_VEL
LIN {X 0,Y 355.465,Z 557.03,A -85,B 0,C 180,E1 12275.974,E2 12275.974} C_VEL
LIN {X 0,Y 355.384,Z 557.03,A -85,B 0,C 180,E1 12280.176,E2 12280.176} C_VEL
LIN {X 0,Y 357.781,Z 562.655,A -85,B 0,C 180,E1 12280.852,E2 12280.852} C_VEL
LIN {X 0,Y 376.081,Z 590.986,A -85,B 0,C 180,E1 12284.99,E2 12284.99} C_VEL
LIN {X 0,Y 391.37,Z 622.078,A -85,B 0,C 180,E1 12288.641,E2 12288.641} C_VEL
LIN {X 0,Y 396.991,Z 637.263,A -85,B 0,C 180,E1 12290.313,E2 12290.313} C_VEL
LIN {X 0,Y 391.23,Z 672.856,A -85,B 0,C 180,E1 12292.462,E2 12292.462} C_VEL
LIN {X 0,Y 383.82,Z 707.252,A -85,B 0,C 180,E1 12295.588,E2 12295.588} C_VEL
LIN {X 0,Y 376.428,Z 736.05,A -85,B 0,C 180,E1 12299.327,E2 12299.327} C_VEL
LIN {X 0,Y 369.55,Z 760.678,A -85,B 0,C 180,E1 12303.747,E2 12303.747} C_VEL
LIN {X 0,Y 363.742,Z 781.775,A -85,B 0,C 180,E1 12309.044,E2 12309.044} C_VEL
LIN {X 0,Y 360.129,Z 797.454,A -85,B 0,C 180,E1 12314.766,E2 12314.766} C_VEL
LIN {X 0,Y 358.356,Z 807.19,A -85,B 0,C 180,E1 12320.27,E2 12320.27} C_VEL
LIN {X 0,Y 357.665,Z 812.004,A -85,B 0,C 180,E1 12325.143,E2 12325.143} C_VEL
LIN {X 0,Y 357.527,Z 813.633,A -85,B 0,C 180,E1 12330,E2 12330} C_VEL
LIN {X 0,Y 357.803,Z 810.934,A -85,B 0,C 180,E1 12336.194,E2 12336.194} C_VEL
LIN {X 0,Y 358.924,Z 803.233,A -85,B 0,C 180,E1 12342.176,E2 12342.176} C_VEL
LIN {X 0,Y 361.435,Z 791.213,A -85,B 0,C 180,E1 12347.68,E2 12347.68} C_VEL
LIN {X 0,Y 366.018,Z 773.563,A -85,B 0,C 180,E1 12353.139,E2 12353.139} C_VEL
LIN {X 0,Y 372.476,Z 750.325,A -85,B 0,C 180,E1 12358.199,E2 12358.199} C_VEL
LIN {X 0,Y 380.056,Z 722.167,A -85,B 0,C 180,E1 12362.534,E2 12362.534} C_VEL
LIN {X 0,Y 387.423,Z 691.487,A -85,B 0,C 180,E1 12365.887,E2 12365.887} C_VEL
LIN {X 0,Y 393.756,Z 658.926,A -85,B 0,C 180,E1 12368.385,E2 12368.385} C_VEL
LIN {X 0,Y 396.895,Z 636.557,A -85,B 0,C 180,E1 12369.644,E2 12369.644} C_VEL
LIN {X 0,Y 383.393,Z 604.649,A -85,B 0,C 180,E1 12373.247,E2 12373.247} C_VEL
LIN {X 0,Y 366.133,Z 574.976,A -85,B 0,C 180,E1 12377.081,E2 12377.081} C_VEL
LIN {X 0,Y 357.287,Z 562.054,A -85,B 0,C 180,E1 12379.148,E2 12379.148} C_VEL
LIN {X 0,Y 355.424,Z 557.03,A -85,B 0,C 180,E1 12379.815,E2 12379.815} C_VEL
LIN {X 0,Y 355.502,Z 557.03,A -85,B 0,C 180,E1 12386.385,E2 12386.385} C_VEL
LIN {X 0,Y 355.752,Z 557.03,A -85,B 0,C 180,E1 12393.346,E2 12393.346} C_VEL
LIN {X 0,Y 356.103,Z 557.03,A -85,B 0,C 180,E1 12400.117,E2 12400.117} C_VEL
LIN {X 0,Y 356.468,Z 557.03,A -85,B 0,C 180,E1 12407.74,E2 12407.74} C_VEL
LIN {X 0,Y 356.904,Z 557.03,A -85,B 0,C 180,E1 12415.134,E2 12415.134} C_VEL
LIN {X 0,Y 357.074,Z 557.03,A -85,B 0,C 180,E1 12422.43,E2 12422.43} C_VEL
LIN {X 0,Y 356.492,Z 557.03,A -85,B 0,C 180,E1 12429.781,E2 12429.781} C_VEL
LIN {X 0,Y 356.182,Z 557.03,A -85,B 0,C 180,E1 12437.31,E2 12437.31} C_VEL
LIN {X 0,Y 355.778,Z 557.03,A -85,B 0,C 180,E1 12445.185,E2 12445.185} C_VEL
LIN {X 0,Y 355.517,Z 557.03,A -85,B 0,C 180,E1 12451.599,E2 12451.599} C_VEL
LIN {X 0,Y 355.489,Z 557.03,A -85,B 0,C 180,E1 12455.8,E2 12455.8} C_VEL
LIN {X 0,Y 357.954,Z 562.791,A -85,B 0,C 180,E1 12456.514,E2 12456.514} C_VEL
LIN {X 0,Y 374.113,Z 588.149,A -85,B 0,C 180,E1 12460.243,E2 12460.243} C_VEL
LIN {X 0,Y 389.634,Z 618.118,A -85,B 0,C 180,E1 12463.702,E2 12463.702} C_VEL
LIN {X 0,Y 397.802,Z 642.06,A -85,B 0,C 180,E1 12466.041,E2 12466.041} C_VEL
LIN {X 0,Y 391.757,Z 681.635,A -85,B 0,C 180,E1 12468.19,E2 12468.19} C_VEL
LIN {X 0,Y 384.491,Z 718.58,A -85,B 0,C 180,E1 12471.21,E2 12471.21} C_VEL
LIN {X 0,Y 376.8,Z 752.241,A -85,B 0,C 180,E1 12475.069,E2 12475.069} C_VEL
LIN {X 0,Y 369.948,Z 780.869,A -85,B 0,C 180,E1 12479.529,E2 12479.529} C_VEL
LIN {X 0,Y 364.191,Z 805.908,A -85,B 0,C 180,E1 12484.779,E2 12484.779} C_VEL
LIN {X 0,Y 360.422,Z 825.454,A -85,B 0,C 180,E1 12490.363,E2 12490.363} C_VEL
LIN {X 0,Y 358.237,Z 840.343,A -85,B 0,C 180,E1 12496.412,E2 12496.412} C_VEL
LIN {X 0,Y 357.545,Z 848.505,A -85,B 0,C 180,E1 12501.477,E2 12501.477} C_VEL
LIN {X 0,Y 357.318,Z 853.29,A -85,B 0,C 180,E1 12507.572,E2 12507.572} C_VEL
LIN {X 0,Y 357.338,Z 853.292,A -85,B 0,C 180,E1 12512.429,E2 12512.429} C_VEL
LIN {X 0,Y 357.545,Z 848.51,A -85,B 0,C 180,E1 12518.524,E2 12518.524} C_VEL
LIN {X 0,Y 358.014,Z 842.92,A -85,B 0,C 180,E1 12522.234,E2 12522.234} C_VEL
LIN {X 0,Y 355.912,Z 839.148,A -85,B 0,C 180,E1 12524.227,E2 12524.227} C_VEL
LIN {X 0,Y 351.489,Z 832.724,A -85,B 0,C 180,E1 12527.19,E2 12527.19} C_VEL
LIN {X 0,Y 351.539,Z 831.876,A -85,B 0,C 180,E1 12527.523,E2 12527.523} C_VEL
LIN {X 0,Y 354.933,Z 813.88,A -85,B 0,C 180,E1 12533.532,E2 12533.532} C_VEL
LIN {X 0,Y 360.064,Z 791.646,A -85,B 0,C 180,E1 12538.919,E2 12538.919} C_VEL
LIN {X 0,Y 367.066,Z 763.524,A -85,B 0,C 180,E1 12543.951,E2 12543.951} C_VEL
LIN {X 0,Y 374.8,Z 732.281,A -85,B 0,C 180,E1 12548.057,E2 12548.057} C_VEL
LIN {X 0,Y 382.659,Z 696.814,A -85,B 0,C 180,E1 12551.433,E2 12551.433} C_VEL
LIN {X 0,Y 389.559,Z 658.98,A -85,B 0,C 180,E1 12553.913,E2 12553.913} C_VEL
LIN {X 0,Y 391.312,Z 642.464,A -85,B 0,C 180,E1 12554.789,E2 12554.789} C_VEL
LIN {X 0,Y 380.504,Z 614.081,A -85,B 0,C 180,E1 12557.823,E2 12557.823} C_VEL
LIN {X 0,Y 363.971,Z 583.908,A -85,B 0,C 180,E1 12561.681,E2 12561.681} C_VEL
LIN {X 0,Y 349.885,Z 562.633,A -85,B 0,C 180,E1 12565.194,E2 12565.194} C_VEL
LIN {X 0,Y 347.574,Z 557.03,A -85,B 0,C 180,E1 12565.949,E2 12565.949} C_VEL
LIN {X 0,Y 347.72,Z 557.03,A -85,B 0,C 180,E1 12571.384,E2 12571.384} C_VEL
LIN {X 0,Y 347.939,Z 557.03,A -85,B 0,C 180,E1 12576.945,E2 12576.945} C_VEL
LIN {X 0,Y 348.239,Z 557.03,A -85,B 0,C 180,E1 12583.04,E2 12583.04} C_VEL
LIN {X 0,Y 348.505,Z 557.03,A -85,B 0,C 180,E1 12589.993,E2 12589.993} C_VEL
LIN {X 0,Y 349.162,Z 557.03,A -85,B 0,C 180,E1 12597.514,E2 12597.514} C_VEL
LIN {X 0,Y 348.98,Z 557.03,A -85,B 0,C 180,E1 12604.977,E2 12604.977} C_VEL
LIN {X 0,Y 348.485,Z 557.03,A -85,B 0,C 180,E1 12612.545,E2 12612.545} C_VEL
LIN {X 0,Y 348.287,Z 557.03,A -85,B 0,C 180,E1 12617.714,E2 12617.714} C_VEL
LIN {X 0,Y 347.84,Z 557.03,A -85,B 0,C 180,E1 12625.8,E2 12625.8} C_VEL
LIN {X 0,Y 347.636,Z 557.03,A -85,B 0,C 180,E1 12631.506,E2 12631.506} C_VEL
LIN {X 0,Y 347.416,Z 557.477,A -85,B 0,C 180,E1 12638.491,E2 12638.491} C_VEL
LIN {X 0,Y 349.814,Z 562.671,A -85,B 0,C 180,E1 12639.188,E2 12639.188} C_VEL
LIN {X 0,Y 360.141,Z 577.808,A -85,B 0,C 180,E1 12641.761,E2 12641.761} C_VEL
LIN {X 0,Y 376.867,Z 606.183,A -85,B 0,C 180,E1 12645.685,E2 12645.685} C_VEL
LIN {X 0,Y 390.049,Z 637.55,A -85,B 0,C 180,E1 12649.401,E2 12649.401} C_VEL
LIN {X 0,Y 390.172,Z 644.338,A -85,B 0,C 180,E1 12649.885,E2 12649.885} C_VEL
LIN {X 0,Y 384.136,Z 678.142,A -85,B 0,C 180,E1 12652.105,E2 12652.105} C_VEL
LIN {X 0,Y 376.565,Z 710.601,A -85,B 0,C 180,E1 12655.219,E2 12655.219} C_VEL
LIN {X 0,Y 368.739,Z 739.594,A -85,B 0,C 180,E1 12659.17,E2 12659.17} C_VEL
LIN {X 0,Y 361.521,Z 764.226,A -85,B 0,C 180,E1 12663.844,E2 12663.844} C_VEL
LIN {X 0,Y 355.503,Z 785.218,A -85,B 0,C 180,E1 12669.535,E2 12669.535} C_VEL
LIN {X 0,Y 352.146,Z 799.179,A -85,B 0,C 180,E1 12675.05,E2 12675.05} C_VEL
LIN {X 0,Y 350.238,Z 809.125,A -85,B 0,C 180,E1 12681.297,E2 12681.297} C_VEL
LIN {X 0,Y 349.612,Z 813.658,A -85,B 0,C 180,E1 12687.517,E2 12687.517} C_VEL
LIN {X 0,Y 349.651,Z 813.617,A -85,B 0,C 180,E1 12692.481,E2 12692.481} C_VEL
LIN {X 0,Y 350.271,Z 809.007,A -85,B 0,C 180,E1 12698.701,E2 12698.701} C_VEL
LIN {X 0,Y 352.163,Z 798.986,A -85,B 0,C 180,E1 12704.948,E2 12704.948} C_VEL
LIN {X 0,Y 355.806,Z 784.018,A -85,B 0,C 180,E1 12710.769,E2 12710.769} C_VEL
LIN {X 0,Y 361.669,Z 763.602,A -85,B 0,C 180,E1 12716.193,E2 12716.193} C_VEL
LIN {X 0,Y 369.119,Z 738.135,A -85,B 0,C 180,E1 12720.963,E2 12720.963} C_VEL
LIN {X 0,Y 376.657,Z 710.381,A -85,B 0,C 180,E1 12724.7,E2 12724.7} C_VEL
LIN {X 0,Y 384.056,Z 678.172,A -85,B 0,C 180,E1 12727.799,E2 12727.799} C_VEL
LIN {X 0,Y 390.595,Z 641.72,A -85,B 0,C 180,E1 12730.142,E2 12730.142} C_VEL
LIN {X 0,Y 386.773,Z 628.806,A -85,B 0,C 180,E1 12731.517,E2 12731.517} C_VEL
LIN {X 0,Y 372.019,Z 597.078,A -85,B 0,C 180,E1 12735.383,E2 12735.383} C_VEL
LIN {X 0,Y 354.091,Z 568.72,A -85,B 0,C 180,E1 12739.596,E2 12739.596} C_VEL
LIN {X 0,Y 349.718,Z 562.525,A -85,B 0,C 180,E1 12740.714,E2 12740.714} C_VEL
LIN {X 0,Y 347.418,Z 557.03,A -85,B 0,C 180,E1 12741.442,E2 12741.442} C_VEL
LIN {X 0,Y 347.636,Z 557.03,A -85,B 0,C 180,E1 12748.494,E2 12748.494} C_VEL
LIN {X 0,Y 347.859,Z 557.03,A -85,B 0,C 180,E1 12756.066,E2 12756.066} C_VEL
LIN {X 0,Y 348.384,Z 557.03,A -85,B 0,C 180,E1 12762.959,E2 12762.959} C_VEL
LIN {X 0,Y 348.618,Z 557.03,A -85,B 0,C 180,E1 12769.997,E2 12769.997} C_VEL
LIN {X 0,Y 349.131,Z 557.03,A -85,B 0,C 180,E1 12777.515,E2 12777.515} C_VEL
LIN {X 0,Y 348.968,Z 557.03,A -85,B 0,C 180,E1 12783.73,E2 12783.73} C_VEL
LIN {X 0,Y 348.555,Z 557.03,A -85,B 0,C 180,E1 12790.006,E2 12790.006} C_VEL
LIN {X 0,Y 348.218,Z 557.03,A -85,B 0,C 180,E1 12797.719,E2 12797.719} C_VEL
LIN {X 0,Y 347.835,Z 557.03,A -85,B 0,C 180,E1 12805.802,E2 12805.802} C_VEL
LIN {X 0,Y 347.612,Z 557.03,A -85,B 0,C 180,E1 12813.704,E2 12813.704} C_VEL
LIN {X 0,Y 347.585,Z 557.391,A -85,B 0,C 180,E1 12814.145,E2 12814.145} C_VEL
LIN {X 0,Y 350.005,Z 562.728,A -85,B 0,C 180,E1 12814.865,E2 12814.865} C_VEL
LIN {X 0,Y 365.784,Z 586.696,A -85,B 0,C 180,E1 12818.757,E2 12818.757} C_VEL
LIN {X 0,Y 382.505,Z 618.297,A -85,B 0,C 180,E1 12822.673,E2 12822.673} C_VEL
LIN {X 0,Y 391.593,Z 643.476,A -85,B 0,C 180,E1 12825.317,E2 12825.317} C_VEL
LIN {X 0,Y 385.267,Z 683.354,A -85,B 0,C 180,E1 12827.568,E2 12827.568} C_VEL
LIN {X 0,Y 377.8,Z 719.445,A -85,B 0,C 180,E1 12830.593,E2 12830.593} C_VEL
LIN {X 0,Y 369.826,Z 752.713,A -85,B 0,C 180,E1 12834.492,E2 12834.492} C_VEL
LIN {X 0,Y 362.397,Z 782.206,A -85,B 0,C 180,E1 12839.223,E2 12839.223} C_VEL
LIN {X 0,Y 356.474,Z 806.72,A -85,B 0,C 180,E1 12844.553,E2 12844.553} C_VEL
LIN {X 0,Y 352.432,Z 826.799,A -85,B 0,C 180,E1 12850.558,E2 12850.558} C_VEL
LIN {X 0,Y 350.284,Z 841.231,A -85,B 0,C 180,E1 12856.809,E2 12856.809} C_VEL
LIN {X 0,Y 349.587,Z 849.386,A -85,B 0,C 180,E1 12862.535,E2 12862.535} C_VEL
LIN {X 0,Y 349.421,Z 852.845,A -85,B 0,C 180,E1 12867.517,E2 12867.517} C_VEL
LIN {X 0,Y 349.44,Z 852.848,A -85,B 0,C 180,E1 12872.484,E2 12872.484} C_VEL
LIN {X 0,Y 349.656,Z 848.05,A -85,B 0,C 180,E1 12878.717,E2 12878.717} C_VEL
LIN {X 0,Y 350.733,Z 837.681,A -85,B 0,C 180,E1 12885.012,E2 12885.012} C_VEL
LIN {X 0,Y 351.539,Z 831.876,A -85,B 0,C 180,E1 12887.523,E2 12887.523} C_VEL
LIN {X 0,Y 350.871,Z 828.602,A -85,B 0,C 180,E1 12888.839,E2 12888.839} C_VEL
LIN {X 0,Y 346.235,Z 818.85,A -85,B 0,C 180,E1 12892.419,E2 12892.419} C_VEL
LIN {X 0,Y 346.374,Z 817.828,A -85,B 0,C 180,E1 12892.742,E2 12892.742} C_VEL
LIN {X 0,Y 351.779,Z 795.499,A -85,B 0,C 180,E1 12898.609,E2 12898.609} C_VEL
LIN {X 0,Y 359.278,Z 766.886,A -85,B 0,C 180,E1 12904.064,E2 12904.064} C_VEL
LIN {X 0,Y 367.742,Z 734.297,A -85,B 0,C 180,E1 12908.537,E2 12908.537} C_VEL
LIN {X 0,Y 375.911,Z 699.467,A -85,B 0,C 180,E1 12911.966,E2 12911.966} C_VEL
LIN {X 0,Y 382.783,Z 664.143,A -85,B 0,C 180,E1 12914.403,E2 12914.403} C_VEL
LIN {X 0,Y 385.259,Z 645.504,A -85,B 0,C 180,E1 12915.423,E2 12915.423} C_VEL
LIN {X 0,Y 374.741,Z 617.381,A -85,B 0,C 180,E1 12918.582,E2 12918.582} C_VEL
LIN {X 0,Y 358.462,Z 587.096,A -85,B 0,C 180,E1 12922.618,E2 12922.618} C_VEL
LIN {X 0,Y 342.299,Z 562.883,A -85,B 0,C 180,E1 12926.9,E2 12926.9} C_VEL
LIN {X 0,Y 339.779,Z 558.34,A -85,B 0,C 180,E1 12927.677,E2 12927.677} C_VEL
LIN {X 0,Y 339.68,Z 557.03,A -85,B 0,C 180,E1 12927.875,E2 12927.875} C_VEL
LIN {X 0,Y 339.836,Z 557.03,A -85,B 0,C 180,E1 12933.545,E2 12933.545} C_VEL
LIN {X 0,Y 340.154,Z 557.03,A -85,B 0,C 180,E1 12939.185,E2 12939.185} C_VEL
LIN {X 0,Y 340.393,Z 557.03,A -85,B 0,C 180,E1 12947.151,E2 12947.151} C_VEL
LIN {X 0,Y 341.004,Z 557.03,A -85,B 0,C 180,E1 12954.905,E2 12954.905} C_VEL
LIN {X 0,Y 341.352,Z 557.03,A -85,B 0,C 180,E1 12960,E2 12960} C_VEL
LIN {X 0,Y 340.796,Z 557.03,A -85,B 0,C 180,E1 12967.658,E2 12967.658} C_VEL
LIN {X 0,Y 340.402,Z 557.03,A -85,B 0,C 180,E1 12975.476,E2 12975.476} C_VEL
LIN {X 0,Y 340.148,Z 557.03,A -85,B 0,C 180,E1 12980.858,E2 12980.858} C_VEL
LIN {X 0,Y 339.784,Z 557.03,A -85,B 0,C 180,E1 12989.348,E2 12989.348} C_VEL
LIN {X 0,Y 339.436,Z 557.03,A -85,B 0,C 180,E1 12996.592,E2 12996.592} C_VEL
LIN {X 0,Y 341.538,Z 562.31,A -85,B 0,C 180,E1 12997.292,E2 12997.292} C_VEL
LIN {X 0,Y 344.364,Z 566.002,A -85,B 0,C 180,E1 12998.078,E2 12998.078} C_VEL
LIN {X 0,Y 360.746,Z 590.853,A -85,B 0,C 180,E1 13002.282,E2 13002.282} C_VEL
LIN {X 0,Y 376.024,Z 619.98,A -85,B 0,C 180,E1 13006.234,E2 13006.234} C_VEL
LIN {X 0,Y 384.399,Z 644.025,A -85,B 0,C 180,E1 13009.063,E2 13009.063} C_VEL
LIN {X 0,Y 377.949,Z 678.844,A -85,B 0,C 180,E1 13011.371,E2 13011.371} C_VEL
LIN {X 0,Y 370.114,Z 711.196,A -85,B 0,C 180,E1 13014.522,E2 13014.522} C_VEL
LIN {X 0,Y 362.03,Z 739.855,A -85,B 0,C 180,E1 13018.482,E2 13018.482} C_VEL
LIN {X 0,Y 354.351,Z 764.789,A -85,B 0,C 180,E1 13023.288,E2 13023.288} C_VEL
LIN {X 0,Y 348.039,Z 785.69,A -85,B 0,C 180,E1 13029.076,E2 13029.076} C_VEL
LIN {X 0,Y 344.441,Z 799.638,A -85,B 0,C 180,E1 13034.707,E2 13034.707} C_VEL
LIN {X 0,Y 342.405,Z 809.573,A -85,B 0,C 180,E1 13041.096,E2 13041.096} C_VEL
LIN {X 0,Y 341.747,Z 814.1,A -85,B 0,C 180,E1 13047.46,E2 13047.46} C_VEL
LIN {X 0,Y 341.783,Z 814.06,A -85,B 0,C 180,E1 13052.538,E2 13052.538} C_VEL
LIN {X 0,Y 342.438,Z 809.457,A -85,B 0,C 180,E1 13058.902,E2 13058.902} C_VEL
LIN {X 0,Y 344.451,Z 799.448,A -85,B 0,C 180,E1 13065.291,E2 13065.291} C_VEL
LIN {X 0,Y 348.731,Z 783.193,A -85,B 0,C 180,E1 13071.656,E2 13071.656} C_VEL
LIN {X 0,Y 354.909,Z 762.923,A -85,B 0,C 180,E1 13077.02,E2 13077.02} C_VEL
LIN {X 0,Y 362.693,Z 737.458,A -85,B 0,C 180,E1 13081.804,E2 13081.804} C_VEL
LIN {X 0,Y 370.951,Z 708.021,A -85,B 0,C 180,E1 13085.744,E2 13085.744} C_VEL
LIN {X 0,Y 378.957,Z 673.825,A -85,B 0,C 180,E1 13088.927,E2 13088.927} C_VEL
LIN {X 0,Y 384.462,Z 642.26,A -85,B 0,C 180,E1 13090.953,E2 13090.953} C_VEL
LIN {X 0,Y 371.787,Z 610.972,A -85,B 0,C 180,E1 13094.815,E2 13094.815} C_VEL
LIN {X 0,Y 355.26,Z 581.73,A -85,B 0,C 180,E1 13098.964,E2 13098.964} C_VEL
LIN {X 0,Y 342.231,Z 562.946,A -85,B 0,C 180,E1 13102.397,E2 13102.397} C_VEL
LIN {X 0,Y 339.606,Z 558.475,A -85,B 0,C 180,E1 13103.181,E2 13103.181} C_VEL
LIN {X 0,Y 339.459,Z 557.03,A -85,B 0,C 180,E1 13103.401,E2 13103.401} C_VEL
LIN {X 0,Y 339.793,Z 557.03,A -85,B 0,C 180,E1 13110.653,E2 13110.653} C_VEL
LIN {X 0,Y 340.153,Z 557.03,A -85,B 0,C 180,E1 13119.183,E2 13119.183} C_VEL
LIN {X 0,Y 340.63,Z 557.03,A -85,B 0,C 180,E1 13127.161,E2 13127.161} C_VEL
LIN {X 0,Y 341.051,Z 557.03,A -85,B 0,C 180,E1 13134.907,E2 13134.907} C_VEL
LIN {X 0,Y 341.358,Z 557.03,A -85,B 0,C 180,E1 13140,E2 13140} C_VEL
LIN {X 0,Y 340.847,Z 557.03,A -85,B 0,C 180,E1 13147.658,E2 13147.658} C_VEL
LIN {X 0,Y 340.358,Z 557.03,A -85,B 0,C 180,E1 13155.48,E2 13155.48} C_VEL
LIN {X 0,Y 340.11,Z 557.03,A -85,B 0,C 180,E1 13160.862,E2 13160.862} C_VEL
LIN {X 0,Y 339.78,Z 557.03,A -85,B 0,C 180,E1 13169.349,E2 13169.349} C_VEL
LIN {X 0,Y 339.685,Z 557.03,A -85,B 0,C 180,E1 13172.257,E2 13172.257} C_VEL
LIN {X 0,Y 342.001,Z 562.627,A -85,B 0,C 180,E1 13173.052,E2 13173.052} C_VEL
LIN {X 0,Y 349.463,Z 573.604,A -85,B 0,C 180,E1 13175.126,E2 13175.126} C_VEL
LIN {X 0,Y 365.372,Z 599.01,A -85,B 0,C 180,E1 13179.095,E2 13179.095} C_VEL
LIN {X 0,Y 379.171,Z 627.604,A -85,B 0,C 180,E1 13182.651,E2 13182.651} C_VEL
LIN {X 0,Y 385.36,Z 647.14,A -85,B 0,C 180,E1 13184.715,E2 13184.715} C_VEL
LIN {X 0,Y 378.925,Z 684.54,A -85,B 0,C 180,E1 13186.888,E2 13186.888} C_VEL
LIN {X 0,Y 371.108,Z 720.534,A -85,B 0,C 180,E1 13189.976,E2 13189.976} C_VEL
LIN {X 0,Y 362.906,Z 753.193,A -85,B 0,C 180,E1 13193.893,E2 13193.893} C_VEL
LIN {X 0,Y 355.037,Z 782.859,A -85,B 0,C 180,E1 13198.773,E2 13198.773} C_VEL
LIN {X 0,Y 348.517,Z 808.477,A -85,B 0,C 180,E1 13204.556,E2 13204.556} C_VEL
LIN {X 0,Y 344.506,Z 827.642,A -85,B 0,C 180,E1 13210.583,E2 13210.583} C_VEL
LIN {X 0,Y 342.29,Z 842.029,A -85,B 0,C 180,E1 13217.223,E2 13217.223} C_VEL
LIN {X 0,Y 341.567,Z 850.159,A -85,B 0,C 180,E1 13223.638,E2 13223.638} C_VEL
LIN {X 0,Y 341.652,Z 852.87,A -85,B 0,C 180,E1 13230,E2 13230} C_VEL
LIN {X 0,Y 341.571,Z 850.165,A -85,B 0,C 180,E1 13236.363,E2 13236.363} C_VEL
LIN {X 0,Y 342.333,Z 842.034,A -85,B 0,C 180,E1 13242.776,E2 13242.776} C_VEL
LIN {X 0,Y 344.471,Z 827.67,A -85,B 0,C 180,E1 13249.413,E2 13249.413} C_VEL
LIN {X 0,Y 346.374,Z 817.828,A -85,B 0,C 180,E1 13252.742,E2 13252.742} C_VEL
LIN {X 0,Y 344.554,Z 809.834,A -85,B 0,C 180,E1 13255.314,E2 13255.314} C_VEL
LIN {X 0,Y 342.968,Z 801.004,A -85,B 0,C 180,E1 13257.838,E2 13257.838} C_VEL
LIN {X 0,Y 350.316,Z 774.339,A -85,B 0,C 180,E1 13263.425,E2 13263.425} C_VEL
LIN {X 0,Y 358.732,Z 743.608,A -85,B 0,C 180,E1 13268.117,E2 13268.117} C_VEL
LIN {X 0,Y 367.258,Z 710.55,A -85,B 0,C 180,E1 13271.756,E2 13271.756} C_VEL
LIN {X 0,Y 374.817,Z 675.183,A -85,B 0,C 180,E1 13274.541,E2 13274.541} C_VEL
LIN {X 0,Y 379.056,Z 647.985,A -85,B 0,C 180,E1 13276.123,E2 13276.123} C_VEL
LIN {X 0,Y 368.326,Z 618.938,A -85,B 0,C 180,E1 13279.559,E2 13279.559} C_VEL
LIN {X 0,Y 353.008,Z 590.709,A -85,B 0,C 180,E1 13283.578,E2 13283.578} C_VEL
LIN {X 0,Y 338.105,Z 568.303,A -85,B 0,C 180,E1 13287.708,E2 13287.708} C_VEL
LIN {X 0,Y 334.598,Z 563.105,A -85,B 0,C 180,E1 13288.796,E2 13288.796} C_VEL
LIN {X 0,Y 331.873,Z 558.323,A -85,B 0,C 180,E1 13289.71,E2 13289.71} C_VEL
LIN {X 0,Y 331.816,Z 557.03,A -85,B 0,C 180,E1 13290.108,E2 13290.108} C_VEL
LIN {X 0,Y 332.153,Z 557.03,A -85,B 0,C 180,E1 13298.614,E2 13298.614} C_VEL
LIN {X 0,Y 332.352,Z 557.03,A -85,B 0,C 180,E1 13304.138,E2 13304.138} C_VEL
LIN {X 0,Y 332.9,Z 557.03,A -85,B 0,C 180,E1 13312.158,E2 13312.158} C_VEL
LIN {X 0,Y 333.45,Z 557.03,A -85,B 0,C 180,E1 13320,E2 13320} C_VEL
LIN {X 0,Y 332.875,Z 557.03,A -85,B 0,C 180,E1 13327.842,E2 13327.842} C_VEL
LIN {X 0,Y 332.442,Z 557.03,A -85,B 0,C 180,E1 13335.857,E2 13335.857} C_VEL
LIN {X 0,Y 332.152,Z 557.03,A -85,B 0,C 180,E1 13341.385,E2 13341.385} C_VEL
LIN {X 0,Y 331.809,Z 557.03,A -85,B 0,C 180,E1 13349.89,E2 13349.89} C_VEL
LIN {X 0,Y 331.547,Z 557.119,A -85,B 0,C 180,E1 13354.556,E2 13354.556} C_VEL
LIN {X 0,Y 333.714,Z 562.435,A -85,B 0,C 180,E1 13355.335,E2 13355.335} C_VEL
LIN {X 0,Y 336.697,Z 566.271,A -85,B 0,C 180,E1 13356.24,E2 13356.24} C_VEL
LIN {X 0,Y 352.242,Z 589.179,A -85,B 0,C 180,E1 13360.547,E2 13360.547} C_VEL
LIN {X 0,Y 367.445,Z 617.051,A -85,B 0,C 180,E1 13364.668,E2 13364.668} C_VEL
LIN {X 0,Y 378.392,Z 645.746,A -85,B 0,C 180,E1 13368.334,E2 13368.334} C_VEL
LIN {X 0,Y 371.516,Z 680.989,A -85,B 0,C 180,E1 13370.737,E2 13370.737} C_VEL
LIN {X 0,Y 363.35,Z 713.026,A -85,B 0,C 180,E1 13373.943,E2 13373.943} C_VEL
LIN {X 0,Y 354.682,Z 742.255,A -85,B 0,C 180,E1 13378.112,E2 13378.112} C_VEL
LIN {X 0,Y 346.571,Z 767.3,A -85,B 0,C 180,E1 13383.189,E2 13383.189} C_VEL
LIN {X 0,Y 340.648,Z 785.861,A -85,B 0,C 180,E1 13388.488,E2 13388.488} C_VEL
LIN {X 0,Y 336.76,Z 800.095,A -85,B 0,C 180,E1 13394.35,E2 13394.35} C_VEL
LIN {X 0,Y 334.566,Z 810.022,A -85,B 0,C 180,E1 13400.886,E2 13400.886} C_VEL
LIN {X 0,Y 333.858,Z 814.543,A -85,B 0,C 180,E1 13407.4,E2 13407.4} C_VEL
LIN {X 0,Y 333.893,Z 814.503,A -85,B 0,C 180,E1 13412.598,E2 13412.598} C_VEL
LIN {X 0,Y 334.6,Z 809.907,A -85,B 0,C 180,E1 13419.112,E2 13419.112} C_VEL
LIN {X 0,Y 336.783,Z 799.906,A -85,B 0,C 180,E1 13425.648,E2 13425.648} C_VEL
LIN {X 0,Y 341.329,Z 783.673,A -85,B 0,C 180,E1 13432.15,E2 13432.15} C_VEL
LIN {X 0,Y 348.176,Z 762.297,A -85,B 0,C 180,E1 13437.869,E2 13437.869} C_VEL
LIN {X 0,Y 355.962,Z 738.005,A -85,B 0,C 180,E1 13442.478,E2 13442.478} C_VEL
LIN {X 0,Y 364.569,Z 708.622,A -85,B 0,C 180,E1 13446.469,E2 13446.469} C_VEL
LIN {X 0,Y 372.758,Z 675.105,A -85,B 0,C 180,E1 13449.649,E2 13449.649} C_VEL
LIN {X 0,Y 378.238,Z 644.988,A -85,B 0,C 180,E1 13451.643,E2 13451.643} C_VEL
LIN {X 0,Y 366.075,Z 614.267,A -85,B 0,C 180,E1 13455.607,E2 13455.607} C_VEL
LIN {X 0,Y 350.691,Z 586.713,A -85,B 0,C 180,E1 13459.744,E2 13459.744} C_VEL
LIN {X 0,Y 334.795,Z 563.391,A -85,B 0,C 180,E1 13464.218,E2 13464.218} C_VEL
LIN {X 0,Y 331.682,Z 558.36,A -85,B 0,C 180,E1 13465.228,E2 13465.228} C_VEL
LIN {X 0,Y 331.55,Z 557.03,A -85,B 0,C 180,E1 13465.377,E2 13465.377} C_VEL
LIN {X 0,Y 331.908,Z 557.03,A -85,B 0,C 180,E1 13472.863,E2 13472.863} C_VEL
LIN {X 0,Y 332.357,Z 557.03,A -85,B 0,C 180,E1 13481.406,E2 13481.406} C_VEL
LIN {X 0,Y 332.756,Z 557.03,A -85,B 0,C 180,E1 13489.515,E2 13489.515} C_VEL
LIN {X 0,Y 333.339,Z 557.03,A -85,B 0,C 180,E1 13497.397,E2 13497.397} C_VEL
LIN {X 0,Y 333.344,Z 557.03,A -85,B 0,C 180,E1 13502.604,E2 13502.604} C_VEL
LIN {X 0,Y 332.673,Z 557.03,A -85,B 0,C 180,E1 13510.489,E2 13510.489} C_VEL
LIN {X 0,Y 332.272,Z 557.03,A -85,B 0,C 180,E1 13518.6,E2 13518.6} C_VEL
LIN {X 0,Y 331.892,Z 557.03,A -85,B 0,C 180,E1 13527.14,E2 13527.14} C_VEL
LIN {X 0,Y 331.784,Z 557.03,A -85,B 0,C 180,E1 13530.214,E2 13530.214} C_VEL
LIN {X 0,Y 333.862,Z 562.421,A -85,B 0,C 180,E1 13531.024,E2 13531.024} C_VEL
LIN {X 0,Y 336.684,Z 565.918,A -85,B 0,C 180,E1 13531.886,E2 13531.886} C_VEL
LIN {X 0,Y 354.974,Z 593.714,A -85,B 0,C 180,E1 13536.949,E2 13536.949} C_VEL
LIN {X 0,Y 370.244,Z 623.418,A -85,B 0,C 180,E1 13541.026,E2 13541.026} C_VEL
LIN {X 0,Y 379.186,Z 648.542,A -85,B 0,C 180,E1 13543.948,E2 13543.948} C_VEL
LIN {X 0,Y 372.391,Z 686.967,A -85,B 0,C 180,E1 13546.277,E2 13546.277} C_VEL
LIN {X 0,Y 364.462,Z 721.589,A -85,B 0,C 180,E1 13549.331,E2 13549.331} C_VEL
LIN {X 0,Y 356.004,Z 753.677,A -85,B 0,C 180,E1 13553.269,E2 13553.269} C_VEL
LIN {X 0,Y 347.762,Z 783.353,A -85,B 0,C 180,E1 13558.274,E2 13558.274} C_VEL
LIN {X 0,Y 340.783,Z 809.282,A -85,B 0,C 180,E1 13564.331,E2 13564.331} C_VEL
LIN {X 0,Y 336.44,Z 829.088,A -85,B 0,C 180,E1 13570.906,E2 13570.906} C_VEL
LIN {X 0,Y 334.448,Z 841.563,A -85,B 0,C 180,E1 13576.918,E2 13576.918} C_VEL
LIN {X 0,Y 333.697,Z 849.712,A -85,B 0,C 180,E1 13583.487,E2 13583.487} C_VEL
LIN {X 0,Y 333.761,Z 852.427,A -85,B 0,C 180,E1 13590,E2 13590} C_VEL
LIN {X 0,Y 333.7,Z 849.718,A -85,B 0,C 180,E1 13596.514,E2 13596.514} C_VEL
LIN {X 0,Y 334.49,Z 841.57,A -85,B 0,C 180,E1 13603.081,E2 13603.081} C_VEL
LIN {X 0,Y 336.829,Z 826.904,A -85,B 0,C 180,E1 13609.976,E2 13609.976} C_VEL
LIN {X 0,Y 341.503,Z 806.874,A -85,B 0,C 180,E1 13616.318,E2 13616.318} C_VEL
LIN {X 0,Y 342.968,Z 801.004,A -85,B 0,C 180,E1 13617.838,E2 13617.838} C_VEL
LIN {X 0,Y 341.797,Z 791.622,A -85,B 0,C 180,E1 13620.315,E2 13620.315} C_VEL
LIN {X 0,Y 341.21,Z 781.511,A -85,B 0,C 180,E1 13622.712,E2 13622.712} C_VEL
LIN {X 0,Y 349.204,Z 754.227,A -85,B 0,C 180,E1 13627.374,E2 13627.374} C_VEL
LIN {X 0,Y 358.025,Z 722.435,A -85,B 0,C 180,E1 13631.359,E2 13631.359} C_VEL
LIN {X 0,Y 366.343,Z 687.429,A -85,B 0,C 180,E1 13634.513,E2 13634.513} C_VEL
LIN {X 0,Y 372.989,Z 650.862,A -85,B 0,C 180,E1 13636.807,E2 13636.807} C_VEL
LIN {X 0,Y 362.651,Z 622.204,A -85,B 0,C 180,E1 13640.347,E2 13640.347} C_VEL
LIN {X 0,Y 347.181,Z 593.232,A -85,B 0,C 180,E1 13644.704,E2 13644.704} C_VEL
LIN {X 0,Y 331.438,Z 569.691,A -85,B 0,C 180,E1 13649.363,E2 13649.363} C_VEL
LIN {X 0,Y 326.978,Z 563.289,A -85,B 0,C 180,E1 13650.869,E2 13650.869} C_VEL
LIN {X 0,Y 323.99,Z 558.213,A -85,B 0,C 180,E1 13651.973,E2 13651.973} C_VEL
LIN {X 0,Y 323.907,Z 557.03,A -85,B 0,C 180,E1 13652.134,E2 13652.134} C_VEL
LIN {X 0,Y 324.23,Z 557.03,A -85,B 0,C 180,E1 13659.058,E2 13659.058} C_VEL
LIN {X 0,Y 324.507,Z 557.03,A -85,B 0,C 180,E1 13666.51,E2 13666.51} C_VEL
LIN {X 0,Y 325.149,Z 557.03,A -85,B 0,C 180,E1 13674.656,E2 13674.656} C_VEL
LIN {X 0,Y 325.564,Z 557.03,A -85,B 0,C 180,E1 13680,E2 13680} C_VEL
LIN {X 0,Y 324.936,Z 557.03,A -85,B 0,C 180,E1 13688.034,E2 13688.034} C_VEL
LIN {X 0,Y 324.51,Z 557.03,A -85,B 0,C 180,E1 13696.255,E2 13696.255} C_VEL
LIN {X 0,Y 324.178,Z 557.03,A -85,B 0,C 180,E1 13701.938,E2 13701.938} C_VEL
LIN {X 0,Y 323.905,Z 557.03,A -85,B 0,C 180,E1 13707.865,E2 13707.865} C_VEL
LIN {X 0,Y 323.655,Z 557.03,A -85,B 0,C 180,E1 13712.247,E2 13712.247} C_VEL
LIN {X 0,Y 325.713,Z 562.316,A -85,B 0,C 180,E1 13713.105,E2 13713.105} C_VEL
LIN {X 0,Y 328.648,Z 565.688,A -85,B 0,C 180,E1 13714.083,E2 13714.083} C_VEL
LIN {X 0,Y 345.225,Z 589.933,A -85,B 0,C 180,E1 13719.079,E2 13719.079} C_VEL
LIN {X 0,Y 360.856,Z 618.377,A -85,B 0,C 180,E1 13723.584,E2 13723.584} C_VEL
LIN {X 0,Y 372.008,Z 647.616,A -85,B 0,C 180,E1 13727.528,E2 13727.528} C_VEL
LIN {X 0,Y 365.44,Z 681.683,A -85,B 0,C 180,E1 13729.954,E2 13729.954} C_VEL
LIN {X 0,Y 356.982,Z 713.616,A -85,B 0,C 180,E1 13733.196,E2 13733.196} C_VEL
LIN {X 0,Y 347.967,Z 742.783,A -85,B 0,C 180,E1 13737.421,E2 13737.421} C_VEL
LIN {X 0,Y 339.647,Z 767.27,A -85,B 0,C 180,E1 13742.452,E2 13742.452} C_VEL
LIN {X 0,Y 333.246,Z 786.328,A -85,B 0,C 180,E1 13747.986,E2 13747.986} C_VEL
LIN {X 0,Y 329.068,Z 800.553,A -85,B 0,C 180,E1 13753.974,E2 13753.974} C_VEL
LIN {X 0,Y 326.758,Z 810.468,A -85,B 0,C 180,E1 13760.666,E2 13760.666} C_VEL
LIN {X 0,Y 325.97,Z 814.986,A -85,B 0,C 180,E1 13767.337,E2 13767.337} C_VEL
LIN {X 0,Y 326.025,Z 814.946,A -85,B 0,C 180,E1 13772.661,E2 13772.661} C_VEL
LIN {X 0,Y 326.791,Z 810.355,A -85,B 0,C 180,E1 13779.332,E2 13779.332} C_VEL
LIN {X 0,Y 329.095,Z 800.366,A -85,B 0,C 180,E1 13786.023,E2 13786.023} C_VEL
LIN {X 0,Y 333.952,Z 784.152,A -85,B 0,C 180,E1 13792.666,E2 13792.666} C_VEL
LIN {X 0,Y 341.13,Z 762.799,A -85,B 0,C 180,E1 13798.497,E2 13798.497} C_VEL
LIN {X 0,Y 349.291,Z 738.536,A -85,B 0,C 180,E1 13803.178,E2 13803.178} C_VEL
LIN {X 0,Y 358.242,Z 709.219,A -85,B 0,C 180,E1 13807.221,E2 13807.221} C_VEL
LIN {X 0,Y 366.827,Z 675.456,A -85,B 0,C 180,E1 13810.463,E2 13810.463} C_VEL
LIN {X 0,Y 372.14,Z 648.065,A -85,B 0,C 180,E1 13812.305,E2 13812.305} C_VEL
LIN {X 0,Y 360.501,Z 617.754,A -85,B 0,C 180,E1 13816.401,E2 13816.401} C_VEL
LIN {X 0,Y 344.704,Z 588.896,A -85,B 0,C 180,E1 13820.952,E2 13820.952} C_VEL
LIN {X 0,Y 327.193,Z 563.607,A -85,B 0,C 180,E1 13826.273,E2 13826.273} C_VEL
LIN {X 0,Y 323.821,Z 558.626,A -85,B 0,C 180,E1 13827.47,E2 13827.47} C_VEL
LIN {X 0,Y 323.656,Z 557.03,A -85,B 0,C 180,E1 13827.849,E2 13827.849} C_VEL
LIN {X 0,Y 324.013,Z 557.03,A -85,B 0,C 180,E1 13835.133,E2 13835.133} C_VEL
LIN {X 0,Y 324.364,Z 557.03,A -85,B 0,C 180,E1 13840.931,E2 13840.931} C_VEL
LIN {X 0,Y 324.734,Z 557.03,A -85,B 0,C 180,E1 13848.266,E2 13848.266} C_VEL
LIN {X 0,Y 325.203,Z 557.03,A -85,B 0,C 180,E1 13854.658,E2 13854.658} C_VEL
LIN {X 0,Y 325.57,Z 557.03,A -85,B 0,C 180,E1 13860,E2 13860} C_VEL
LIN {X 0,Y 324.969,Z 557.03,A -85,B 0,C 180,E1 13868.035,E2 13868.035} C_VEL
LIN {X 0,Y 324.459,Z 557.03,A -85,B 0,C 180,E1 13876.259,E2 13876.259} C_VEL
LIN {X 0,Y 324.154,Z 557.03,A -85,B 0,C 180,E1 13881.941,E2 13881.941} C_VEL
LIN {X 0,Y 323.916,Z 557.757,A -85,B 0,C 180,E1 13888.034,E2 13888.034} C_VEL
LIN {X 0,Y 326.362,Z 562.803,A -85,B 0,C 180,E1 13888.98,E2 13888.98} C_VEL
LIN {X 0,Y 328.893,Z 565.926,A -85,B 0,C 180,E1 13889.828,E2 13889.828} C_VEL
LIN {X 0,Y 344.666,Z 589.187,A -85,B 0,C 180,E1 13894.631,E2 13894.631} C_VEL
LIN {X 0,Y 360.823,Z 618.18,A -85,B 0,C 180,E1 13899.117,E2 13899.117} C_VEL
LIN {X 0,Y 371.68,Z 646.046,A -85,B 0,C 180,E1 13902.655,E2 13902.655} C_VEL
LIN {X 0,Y 372.801,Z 653.838,A -85,B 0,C 180,E1 13903.397,E2 13903.397} C_VEL
LIN {X 0,Y 365.062,Z 693.181,A -85,B 0,C 180,E1 13905.927,E2 13905.927} C_VEL
LIN {X 0,Y 356.221,Z 729.217,A -85,B 0,C 180,E1 13909.396,E2 13909.396} C_VEL
LIN {X 0,Y 347.4,Z 760.314,A -85,B 0,C 180,E1 13913.556,E2 13913.556} C_VEL
LIN {X 0,Y 339.108,Z 788.485,A -85,B 0,C 180,E1 13918.733,E2 13918.733} C_VEL
LIN {X 0,Y 332.476,Z 812.193,A -85,B 0,C 180,E1 13924.728,E2 13924.728} C_VEL
LIN {X 0,Y 328.39,Z 830.353,A -85,B 0,C 180,E1 13931.172,E2 13931.172} C_VEL
LIN {X 0,Y 326.405,Z 843.302,A -85,B 0,C 180,E1 13938.047,E2 13938.047} C_VEL
LIN {X 0,Y 325.754,Z 850.191,A -85,B 0,C 180,E1 13944.667,E2 13944.667} C_VEL
LIN {X 0,Y 325.885,Z 851.985,A -85,B 0,C 180,E1 13950,E2 13950} C_VEL
LIN {X 0,Y 325.828,Z 849.271,A -85,B 0,C 180,E1 13956.672,E2 13956.672} C_VEL
LIN {X 0,Y 326.662,Z 841.108,A -85,B 0,C 180,E1 13963.4,E2 13963.4} C_VEL
LIN {X 0,Y 328.954,Z 827.421,A -85,B 0,C 180,E1 13970.062,E2 13970.062} C_VEL
LIN {X 0,Y 333.851,Z 807.622,A -85,B 0,C 180,E1 13976.606,E2 13976.606} C_VEL
LIN {X 0,Y 340.761,Z 783.01,A -85,B 0,C 180,E1 13982.419,E2 13982.419} C_VEL
LIN {X 0,Y 341.21,Z 781.511,A -85,B 0,C 180,E1 13982.712,E2 13982.712} C_VEL
LIN {X 0,Y 340.891,Z 770.845,A -85,B 0,C 180,E1 13985.045,E2 13985.045} C_VEL
LIN {X 0,Y 340.492,Z 761.114,A -85,B 0,C 180,E1 13987.046,E2 13987.046} C_VEL
LIN {X 0,Y 340.901,Z 759.57,A -85,B 0,C 180,E1 13987.302,E2 13987.302} C_VEL
LIN {X 0,Y 350.41,Z 727.365,A -85,B 0,C 180,E1 13991.631,E2 13991.631} C_VEL
LIN {X 0,Y 359.707,Z 690.65,A -85,B 0,C 180,E1 13995.118,E2 13995.118} C_VEL
LIN {X 0,Y 366.838,Z 653.2,A -85,B 0,C 180,E1 13997.576,E2 13997.576} C_VEL
LIN {X 0,Y 356.521,Z 624.444,A -85,B 0,C 180,E1 14001.319,E2 14001.319} C_VEL
LIN {X 0,Y 342.344,Z 597.685,A -85,B 0,C 180,E1 14005.582,E2 14005.582} C_VEL
LIN {X 0,Y 327.968,Z 575.788,A -85,B 0,C 180,E1 14010.058,E2 14010.058} C_VEL
LIN {X 0,Y 319.437,Z 563.521,A -85,B 0,C 180,E1 14013.153,E2 14013.153} C_VEL
LIN {X 0,Y 316.196,Z 558.582,A -85,B 0,C 180,E1 14014.474,E2 14014.474} C_VEL
LIN {X 0,Y 316.061,Z 557.03,A -85,B 0,C 180,E1 14014.759,E2 14014.759} C_VEL
LIN {X 0,Y 316.44,Z 557.03,A -85,B 0,C 180,E1 14023.124,E2 14023.124} C_VEL
LIN {X 0,Y 316.999,Z 557.03,A -85,B 0,C 180,E1 14031.762,E2 14031.762} C_VEL
LIN {X 0,Y 317.682,Z 557.03,A -85,B 0,C 180,E1 14040,E2 14040} C_VEL
LIN {X 0,Y 316.995,Z 557.03,A -85,B 0,C 180,E1 14048.237,E2 14048.237} C_VEL
LIN {X 0,Y 316.533,Z 557.03,A -85,B 0,C 180,E1 14056.676,E2 14056.676} C_VEL
LIN {X 0,Y 316.092,Z 557.03,A -85,B 0,C 180,E1 14064.482,E2 14064.482} C_VEL
LIN {X 0,Y 315.813,Z 557.544,A -85,B 0,C 180,E1 14069.738,E2 14069.738} C_VEL
LIN {X 0,Y 318.173,Z 562.644,A -85,B 0,C 180,E1 14070.773,E2 14070.773} C_VEL
LIN {X 0,Y 321.094,Z 566.022,A -85,B 0,C 180,E1 14071.859,E2 14071.859} C_VEL
LIN {X 0,Y 335.152,Z 586.209,A -85,B 0,C 180,E1 14076.562,E2 14076.562} C_VEL
LIN {X 0,Y 350.215,Z 611.476,A -85,B 0,C 180,E1 14081.14,E2 14081.14} C_VEL
LIN {X 0,Y 362.236,Z 639.272,A -85,B 0,C 180,E1 14085.275,E2 14085.275} C_VEL
LIN {X 0,Y 366.046,Z 652.191,A -85,B 0,C 180,E1 14086.984,E2 14086.984} C_VEL
LIN {X 0,Y 358.328,Z 687.267,A -85,B 0,C 180,E1 14089.577,E2 14089.577} C_VEL
LIN {X 0,Y 349.154,Z 719.267,A -85,B 0,C 180,E1 14093.067,E2 14093.067} C_VEL
LIN {X 0,Y 340.084,Z 746.717,A -85,B 0,C 180,E1 14097.329,E2 14097.329} C_VEL
LIN {X 0,Y 331.655,Z 770.309,A -85,B 0,C 180,E1 14102.469,E2 14102.469} C_VEL
LIN {X 0,Y 325.222,Z 788.656,A -85,B 0,C 180,E1 14108.134,E2 14108.134} C_VEL
LIN {X 0,Y 320.979,Z 802.517,A -85,B 0,C 180,E1 14114.397,E2 14114.397} C_VEL
LIN {X 0,Y 318.928,Z 810.916,A -85,B 0,C 180,E1 14120.435,E2 14120.435} C_VEL
LIN {X 0,Y 318.11,Z 815.428,A -85,B 0,C 180,E1 14127.271,E2 14127.271} C_VEL
LIN {X 0,Y 318.153,Z 815.389,A -85,B 0,C 180,E1 14132.727,E2 14132.727} C_VEL
LIN {X 0,Y 318.959,Z 810.804,A -85,B 0,C 180,E1 14139.563,E2 14139.563} C_VEL
LIN {X 0,Y 321.439,Z 800.824,A -85,B 0,C 180,E1 14146.416,E2 14146.416} C_VEL
LIN {X 0,Y 326.58,Z 784.631,A -85,B 0,C 180,E1 14153.207,E2 14153.207} C_VEL
LIN {X 0,Y 334.138,Z 763.299,A -85,B 0,C 180,E1 14159.15,E2 14159.15} C_VEL
LIN {X 0,Y 342.661,Z 739.072,A -85,B 0,C 180,E1 14163.906,E2 14163.906} C_VEL
LIN {X 0,Y 351.978,Z 709.814,A -85,B 0,C 180,E1 14167.999,E2 14167.999} C_VEL
LIN {X 0,Y 360.963,Z 675.932,A -85,B 0,C 180,E1 14171.291,E2 14171.291} C_VEL
LIN {X 0,Y 365.861,Z 650.48,A -85,B 0,C 180,E1 14173.083,E2 14173.083} C_VEL
LIN {X 0,Y 354.665,Z 620.724,A -85,B 0,C 180,E1 14177.313,E2 14177.313} C_VEL
LIN {X 0,Y 340.224,Z 593.881,A -85,B 0,C 180,E1 14181.772,E2 14181.772} C_VEL
LIN {X 0,Y 324.117,Z 570.214,A -85,B 0,C 180,E1 14186.904,E2 14186.904} C_VEL
LIN {X 0,Y 319.11,Z 563.425,A -85,B 0,C 180,E1 14188.739,E2 14188.739} C_VEL
LIN {X 0,Y 316.01,Z 558.812,A -85,B 0,C 180,E1 14189.979,E2 14189.979} C_VEL
LIN {X 0,Y 315.799,Z 557.03,A -85,B 0,C 180,E1 14190.158,E2 14190.158} C_VEL
LIN {X 0,Y 316.178,Z 557.03,A -85,B 0,C 180,E1 14197.477,E2 14197.477} C_VEL
LIN {X 0,Y 316.598,Z 557.03,A -85,B 0,C 180,E1 14203.327,E2 14203.327} C_VEL
LIN {X 0,Y 317.038,Z 557.03,A -85,B 0,C 180,E1 14211.764,E2 14211.764} C_VEL
LIN {X 0,Y 317.681,Z 557.03,A -85,B 0,C 180,E1 14220,E2 14220} C_VEL
LIN {X 0,Y 317.021,Z 557.03,A -85,B 0,C 180,E1 14228.237,E2 14228.237} C_VEL
LIN {X 0,Y 316.461,Z 557.03,A -85,B 0,C 180,E1 14236.892,E2 14236.892} C_VEL
LIN {X 0,Y 316.028,Z 557.249,A -85,B 0,C 180,E1 14245.466,E2 14245.466} C_VEL
LIN {X 0,Y 317.98,Z 562.269,A -85,B 0,C 180,E1 14246.365,E2 14246.365} C_VEL
LIN {X 0,Y 321.12,Z 565.735,A -85,B 0,C 180,E1 14247.536,E2 14247.536} C_VEL
LIN {X 0,Y 335.504,Z 586.869,A -85,B 0,C 180,E1 14252.402,E2 14252.402} C_VEL
LIN {X 0,Y 350.638,Z 612.443,A -85,B 0,C 180,E1 14256.901,E2 14256.901} C_VEL
LIN {X 0,Y 362.791,Z 640.047,A -85,B 0,C 180,E1 14260.814,E2 14260.814} C_VEL
LIN {X 0,Y 367.045,Z 654.527,A -85,B 0,C 180,E1 14262.572,E2 14262.572} C_VEL
LIN {X 0,Y 358.903,Z 694.006,A -85,B 0,C 180,E1 14265.159,E2 14265.159} C_VEL
LIN {X 0,Y 349.686,Z 729.882,A -85,B 0,C 180,E1 14268.679,E2 14268.679} C_VEL
LIN {X 0,Y 340.54,Z 760.731,A -85,B 0,C 180,E1 14272.898,E2 14272.898} C_VEL
LIN {X 0,Y 332.083,Z 788.075,A -85,B 0,C 180,E1 14278.024,E2 14278.024} C_VEL
LIN {X 0,Y 325.096,Z 811.692,A -85,B 0,C 180,E1 14284.112,E2 14284.112} C_VEL
LIN {X 0,Y 320.68,Z 830.033,A -85,B 0,C 180,E1 14290.772,E2 14290.772} C_VEL
LIN {X 0,Y 318.538,Z 843.017,A -85,B 0,C 180,E1 14297.867,E2 14297.867} C_VEL
LIN {X 0,Y 317.873,Z 849.745,A -85,B 0,C 180,E1 14304.534,E2 14304.534} C_VEL
LIN {X 0,Y 317.942,Z 851.486,A -85,B 0,C 180,E1 14310.476,E2 14310.476} C_VEL
LIN {X 0,Y 317.958,Z 848.824,A -85,B 0,C 180,E1 14316.838,E2 14316.838} C_VEL
LIN {X 0,Y 318.82,Z 840.647,A -85,B 0,C 180,E1 14323.736,E2 14323.736} C_VEL
LIN {X 0,Y 321.385,Z 826.636,A -85,B 0,C 180,E1 14330.691,E2 14330.691} C_VEL
LIN {X 0,Y 326.833,Z 805.853,A -85,B 0,C 180,E1 14337.598,E2 14337.598} C_VEL
LIN {X 0,Y 334.239,Z 781.25,A -85,B 0,C 180,E1 14343.418,E2 14343.418} C_VEL
LIN {X 0,Y 340.901,Z 759.57,A -85,B 0,C 180,E1 14347.302,E2 14347.302} C_VEL
LIN {X 0,Y 341.291,Z 747.766,A -85,B 0,C 180,E1 14349.485,E2 14349.485} C_VEL
LIN {X 0,Y 341.406,Z 736.907,A -85,B 0,C 180,E1 14351.309,E2 14351.309} C_VEL
LIN {X 0,Y 341.845,Z 735.193,A -85,B 0,C 180,E1 14351.525,E2 14351.525} C_VEL
LIN {X 0,Y 351.706,Z 699.378,A -85,B 0,C 180,E1 14355.26,E2 14355.26} C_VEL
LIN {X 0,Y 360.078,Z 662.029,A -85,B 0,C 180,E1 14357.912,E2 14357.912} C_VEL
LIN {X 0,Y 360.776,Z 655.566,A -85,B 0,C 180,E1 14358.366,E2 14358.366} C_VEL
LIN {X 0,Y 350.538,Z 626.865,A -85,B 0,C 180,E1 14362.307,E2 14362.307} C_VEL
LIN {X 0,Y 336.95,Z 600.673,A -85,B 0,C 180,E1 14366.701,E2 14366.701} C_VEL
LIN {X 0,Y 321.229,Z 576.821,A -85,B 0,C 180,E1 14371.977,E2 14371.977} C_VEL
LIN {X 0,Y 315.429,Z 569.115,A -85,B 0,C 180,E1 14374.216,E2 14374.216} C_VEL
LIN {X 0,Y 312.05,Z 563.809,A -85,B 0,C 180,E1 14375.68,E2 14375.68} C_VEL
LIN {X 0,Y 308.504,Z 558.991,A -85,B 0,C 180,E1 14377.301,E2 14377.301} C_VEL
LIN {X 0,Y 308.291,Z 557.03,A -85,B 0,C 180,E1 14377.701,E2 14377.701} C_VEL
LIN {X 0,Y 308.596,Z 557.03,A -85,B 0,C 180,E1 14385.8,E2 14385.8} C_VEL
LIN {X 0,Y 309.298,Z 557.03,A -85,B 0,C 180,E1 14394.381,E2 14394.381} C_VEL
LIN {X 0,Y 309.778,Z 557.03,A -85,B 0,C 180,E1 14399.999,E2 14399.999} C_VEL
LIN {X 0,Y 309.334,Z 557.03,A -85,B 0,C 180,E1 14405.617,E2 14405.617} C_VEL
LIN {X 0,Y 308.734,Z 557.03,A -85,B 0,C 180,E1 14414.192,E2 14414.192} C_VEL
LIN {X 0,Y 308.274,Z 557.03,A -85,B 0,C 180,E1 14421.065,E2 14421.065} C_VEL
LIN {X 0,Y 307.975,Z 557.04,A -85,B 0,C 180,E1 14426.769,E2 14426.769} C_VEL
LIN {X 0,Y 309.641,Z 561.912,A -85,B 0,C 180,E1 14427.688,E2 14427.688} C_VEL
LIN {X 0,Y 313.396,Z 565.954,A -85,B 0,C 180,E1 14429.282,E2 14429.282} C_VEL
LIN {X 0,Y 326.953,Z 584.972,A -85,B 0,C 180,E1 14434.356,E2 14434.356} C_VEL
LIN {X 0,Y 342.753,Z 610.894,A -85,B 0,C 180,E1 14439.527,E2 14439.527} C_VEL
LIN {X 0,Y 354.708,Z 637.832,A -85,B 0,C 180,E1 14443.832,E2 14443.832} C_VEL
LIN {X 0,Y 360.075,Z 654.582,A -85,B 0,C 180,E1 14446.221,E2 14446.221} C_VEL
LIN {X 0,Y 351.805,Z 689.904,A -85,B 0,C 180,E1 14448.935,E2 14448.935} C_VEL
LIN {X 0,Y 342.415,Z 721.198,A -85,B 0,C 180,E1 14452.458,E2 14452.458} C_VEL
LIN {X 0,Y 332.782,Z 748.931,A -85,B 0,C 180,E1 14456.909,E2 14456.909} C_VEL
LIN {X 0,Y 324.119,Z 772.07,A -85,B 0,C 180,E1 14462.151,E2 14462.151} C_VEL
LIN {X 0,Y 316.868,Z 791.847,A -85,B 0,C 180,E1 14468.661,E2 14468.661} C_VEL
LIN {X 0,Y 313.022,Z 803.962,A -85,B 0,C 180,E1 14474.573,E2 14474.573} C_VEL
LIN {X 0,Y 310.806,Z 812.687,A -85,B 0,C 180,E1 14481.596,E2 14481.596} C_VEL
LIN {X 0,Y 310.221,Z 815.871,A -85,B 0,C 180,E1 14487.202,E2 14487.202} C_VEL
LIN {X 0,Y 310.264,Z 815.832,A -85,B 0,C 180,E1 14492.797,E2 14492.797} C_VEL
LIN {X 0,Y 311.137,Z 811.253,A -85,B 0,C 180,E1 14499.806,E2 14499.806} C_VEL
LIN {X 0,Y 313.793,Z 801.282,A -85,B 0,C 180,E1 14506.827,E2 14506.827} C_VEL
LIN {X 0,Y 319.251,Z 785.107,A -85,B 0,C 180,E1 14513.772,E2 14513.772} C_VEL
LIN {X 0,Y 327.214,Z 763.794,A -85,B 0,C 180,E1 14519.828,E2 14519.828} C_VEL
LIN {X 0,Y 336.089,Z 739.604,A -85,B 0,C 180,E1 14524.662,E2 14524.662} C_VEL
LIN {X 0,Y 345.781,Z 710.405,A -85,B 0,C 180,E1 14528.806,E2 14528.806} C_VEL
LIN {X 0,Y 355.191,Z 676.211,A -85,B 0,C 180,E1 14532.165,E2 14532.165} C_VEL
LIN {X 0,Y 359.97,Z 654.027,A -85,B 0,C 180,E1 14533.733,E2 14533.733} C_VEL
LIN {X 0,Y 349.067,Z 623.987,A -85,B 0,C 180,E1 14538.176,E2 14538.176} C_VEL
LIN {X 0,Y 334.916,Z 597.179,A -85,B 0,C 180,E1 14542.902,E2 14542.902} C_VEL
LIN {X 0,Y 320.542,Z 576.154,A -85,B 0,C 180,E1 14547.738,E2 14547.738} C_VEL
LIN {X 0,Y 315.786,Z 569.674,A -85,B 0,C 180,E1 14549.558,E2 14549.558} C_VEL
LIN {X 0,Y 311.938,Z 563.882,A -85,B 0,C 180,E1 14551.19,E2 14551.19} C_VEL
LIN {X 0,Y 308.279,Z 559.17,A -85,B 0,C 180,E1 14552.828,E2 14552.828} C_VEL
LIN {X 0,Y 307.999,Z 557.03,A -85,B 0,C 180,E1 14553.231,E2 14553.231} C_VEL
LIN {X 0,Y 308.401,Z 557.03,A -85,B 0,C 180,E1 14559.902,E2 14559.902} C_VEL
LIN {X 0,Y 308.81,Z 557.03,A -85,B 0,C 180,E1 14565.811,E2 14565.811} C_VEL
LIN {X 0,Y 309.343,Z 557.03,A -85,B 0,C 180,E1 14574.383,E2 14574.383} C_VEL
LIN {X 0,Y 309.777,Z 557.03,A -85,B 0,C 180,E1 14580.001,E2 14580.001} C_VEL
LIN {X 0,Y 309.074,Z 557.03,A -85,B 0,C 180,E1 14588.451,E2 14588.451} C_VEL
LIN {X 0,Y 308.539,Z 557.03,A -85,B 0,C 180,E1 14597.123,E2 14597.123} C_VEL
LIN {X 0,Y 308.265,Z 557.21,A -85,B 0,C 180,E1 14602.577,E2 14602.577} C_VEL
LIN {X 0,Y 310.062,Z 562.122,A -85,B 0,C 180,E1 14603.549,E2 14603.549} C_VEL
LIN {X 0,Y 313.397,Z 565.63,A -85,B 0,C 180,E1 14604.964,E2 14604.964} C_VEL
LIN {X 0,Y 327.266,Z 585.622,A -85,B 0,C 180,E1 14610.205,E2 14610.205} C_VEL
LIN {X 0,Y 343.432,Z 612.325,A -85,B 0,C 180,E1 14615.398,E2 14615.398} C_VEL
LIN {X 0,Y 355.686,Z 639.684,A -85,B 0,C 180,E1 14619.557,E2 14619.557} C_VEL
LIN {X 0,Y 360.876,Z 657.541,A -85,B 0,C 180,E1 14621.837,E2 14621.837} C_VEL
LIN {X 0,Y 352.561,Z 695.784,A -85,B 0,C 180,E1 14624.443,E2 14624.443} C_VEL
LIN {X 0,Y 343.209,Z 730.551,A -85,B 0,C 180,E1 14627.934,E2 14627.934} C_VEL
LIN {X 0,Y 333.526,Z 761.765,A -85,B 0,C 180,E1 14632.313,E2 14632.313} C_VEL
LIN {X 0,Y 324.296,Z 790.131,A -85,B 0,C 180,E1 14637.836,E2 14637.836} C_VEL
LIN {X 0,Y 317.078,Z 813.468,A -85,B 0,C 180,E1 14644.17,E2 14644.17} C_VEL
LIN {X 0,Y 312.661,Z 831.168,A -85,B 0,C 180,E1 14650.994,E2 14650.994} C_VEL
LIN {X 0,Y 310.645,Z 843.021,A -85,B 0,C 180,E1 14657.877,E2 14657.877} C_VEL
LIN {X 0,Y 309.982,Z 849.298,A -85,B 0,C 180,E1 14664.395,E2 14664.395} C_VEL
LIN {X 0,Y 310.128,Z 851.101,A -85,B 0,C 180,E1 14670.001,E2 14670.001} C_VEL
LIN {X 0,Y 310.069,Z 848.377,A -85,B 0,C 180,E1 14677.012,E2 14677.012} C_VEL
LIN {X 0,Y 310.992,Z 840.186,A -85,B 0,C 180,E1 14684.089,E2 14684.089} C_VEL
LIN {X 0,Y 313.776,Z 826.16,A -85,B 0,C 180,E1 14691.217,E2 14691.217} C_VEL
LIN {X 0,Y 319.561,Z 805.347,A -85,B 0,C 180,E1 14698.281,E2 14698.281} C_VEL
LIN {X 0,Y 327.231,Z 781.151,A -85,B 0,C 180,E1 14704.126,E2 14704.126} C_VEL
LIN {X 0,Y 336.334,Z 753.069,A -85,B 0,C 180,E1 14709.068,E2 14709.068} C_VEL
LIN {X 0,Y 341.845,Z 735.193,A -85,B 0,C 180,E1 14711.525,E2 14711.525} C_VEL
LIN {X 0,Y 341.084,Z 726.964,A -85,B 0,C 180,E1 14712.949,E2 14712.949} C_VEL
LIN {X 0,Y 340.356,Z 719.54,A -85,B 0,C 180,E1 14714.182,E2 14714.182} C_VEL
LIN {X 0,Y 340.702,Z 718.33,A -85,B 0,C 180,E1 14714.314,E2 14714.314} C_VEL
LIN {X 0,Y 350.145,Z 682.458,A -85,B 0,C 180,E1 14717.497,E2 14717.497} C_VEL
LIN {X 0,Y 354.742,Z 658.136,A -85,B 0,C 180,E1 14719.149,E2 14719.149} C_VEL
LIN {X 0,Y 344.731,Z 629.486,A -85,B 0,C 180,E1 14723.302,E2 14723.302} C_VEL
LIN {X 0,Y 331.849,Z 604.471,A -85,B 0,C 180,E1 14727.777,E2 14727.777} C_VEL
LIN {X 0,Y 318.152,Z 583.203,A -85,B 0,C 180,E1 14732.645,E2 14732.645} C_VEL
LIN {X 0,Y 309.057,Z 570.513,A -85,B 0,C 180,E1 14736.45,E2 14736.45} C_VEL
LIN {X 0,Y 304.517,Z 563.991,A -85,B 0,C 180,E1 14738.669,E2 14738.669} C_VEL
LIN {X 0,Y 300.72,Z 559.097,A -85,B 0,C 180,E1 14740.707,E2 14740.707} C_VEL
LIN {X 0,Y 300.449,Z 557.03,A -85,B 0,C 180,E1 14741.262,E2 14741.262} C_VEL
LIN {X 0,Y 300.847,Z 557.03,A -85,B 0,C 180,E1 14748.387,E2 14748.387} C_VEL
LIN {X 0,Y 301.693,Z 557.03,A -85,B 0,C 180,E1 14757.123,E2 14757.123} C_VEL
LIN {X 0,Y 301.696,Z 557.03,A -85,B 0,C 180,E1 14762.876,E2 14762.876} C_VEL
LIN {X 0,Y 300.959,Z 557.03,A -85,B 0,C 180,E1 14771.608,E2 14771.608} C_VEL
LIN {X 0,Y 300.597,Z 557.03,A -85,B 0,C 180,E1 14777.588,E2 14777.588} C_VEL
LIN {X 0,Y 300.291,Z 557.769,A -85,B 0,C 180,E1 14783.383,E2 14783.383} C_VEL
LIN {X 0,Y 302.589,Z 562.784,A -85,B 0,C 180,E1 14784.776,E2 14784.776} C_VEL
LIN {X 0,Y 305.62,Z 565.588,A -85,B 0,C 180,E1 14786.256,E2 14786.256} C_VEL
LIN {X 0,Y 310.073,Z 571.367,A -85,B 0,C 180,E1 14788.328,E2 14788.328} C_VEL
LIN {X 0,Y 324.996,Z 593.405,A -85,B 0,C 180,E1 14794.188,E2 14794.188} C_VEL
LIN {X 0,Y 339.021,Z 617.695,A -85,B 0,C 180,E1 14799.144,E2 14799.144} C_VEL
LIN {X 0,Y 350.077,Z 644.242,A -85,B 0,C 180,E1 14803.503,E2 14803.503} C_VEL
LIN {X 0,Y 353.869,Z 658.065,A -85,B 0,C 180,E1 14805.516,E2 14805.516} C_VEL
LIN {X 0,Y 345.864,Z 690.635,A -85,B 0,C 180,E1 14808.084,E2 14808.084} C_VEL
LIN {X 0,Y 336.103,Z 721.917,A -85,B 0,C 180,E1 14811.656,E2 14811.656} C_VEL
LIN {X 0,Y 326.145,Z 749.441,A -85,B 0,C 180,E1 14816.146,E2 14816.146} C_VEL
LIN {X 0,Y 316.496,Z 774.032,A -85,B 0,C 180,E1 14821.881,E2 14821.881} C_VEL
LIN {X 0,Y 309.609,Z 791.87,A -85,B 0,C 180,E1 14827.936,E2 14827.936} C_VEL
LIN {X 0,Y 304.961,Z 805.495,A -85,B 0,C 180,E1 14834.891,E2 14834.891} C_VEL
LIN {X 0,Y 302.971,Z 813.132,A -85,B 0,C 180,E1 14841.377,E2 14841.377} C_VEL
LIN {X 0,Y 302.341,Z 816.314,A -85,B 0,C 180,E1 14847.129,E2 14847.129} C_VEL
LIN {X 0,Y 302.402,Z 816.275,A -85,B 0,C 180,E1 14852.869,E2 14852.869} C_VEL
LIN {X 0,Y 303.335,Z 811.701,A -85,B 0,C 180,E1 14860.06,E2 14860.06} C_VEL
LIN {X 0,Y 306.146,Z 801.739,A -85,B 0,C 180,E1 14867.261,E2 14867.261} C_VEL
LIN {X 0,Y 311.942,Z 785.582,A -85,B 0,C 180,E1 14874.365,E2 14874.365} C_VEL
LIN {X 0,Y 320.315,Z 764.29,A -85,B 0,C 180,E1 14880.538,E2 14880.538} C_VEL
LIN {X 0,Y 329.583,Z 740.135,A -85,B 0,C 180,E1 14885.448,E2 14885.448} C_VEL
LIN {X 0,Y 339.653,Z 710.994,A -85,B 0,C 180,E1 14889.642,E2 14889.642} C_VEL
LIN {X 0,Y 349.312,Z 677.29,A -85,B 0,C 180,E1 14893.004,E2 14893.004} C_VEL
LIN {X 0,Y 353.715,Z 656.294,A -85,B 0,C 180,E1 14894.582,E2 14894.582} C_VEL
LIN {X 0,Y 343.545,Z 627.5,A -85,B 0,C 180,E1 14899.042,E2 14899.042} C_VEL
LIN {X 0,Y 330.279,Z 601.607,A -85,B 0,C 180,E1 14903.832,E2 14903.832} C_VEL
LIN {X 0,Y 314.357,Z 577.659,A -85,B 0,C 180,E1 14909.679,E2 14909.679} C_VEL
LIN {X 0,Y 308.724,Z 570.343,A -85,B 0,C 180,E1 14912.075,E2 14912.075} C_VEL
LIN {X 0,Y 304.459,Z 564.084,A -85,B 0,C 180,E1 14914.146,E2 14914.146} C_VEL
LIN {X 0,Y 300.645,Z 559.663,A -85,B 0,C 180,E1 14916.14,E2 14916.14} C_VEL
LIN {X 0,Y 300.309,Z 557.03,A -85,B 0,C 180,E1 14916.75,E2 14916.75} C_VEL
LIN {X 0,Y 300.84,Z 557.03,A -85,B 0,C 180,E1 14925.427,E2 14925.427} C_VEL
LIN {X 0,Y 301.411,Z 557.03,A -85,B 0,C 180,E1 14934.235,E2 14934.235} C_VEL
LIN {X 0,Y 301.885,Z 557.03,A -85,B 0,C 180,E1 14940.001,E2 14940.001} C_VEL
LIN {X 0,Y 301.371,Z 557.03,A -85,B 0,C 180,E1 14945.767,E2 14945.767} C_VEL
LIN {X 0,Y 300.693,Z 557.03,A -85,B 0,C 180,E1 14954.581,E2 14954.581} C_VEL
LIN {X 0,Y 300.433,Z 557.215,A -85,B 0,C 180,E1 14959.121,E2 14959.121} C_VEL
LIN {X 0,Y 302.32,Z 562.177,A -85,B 0,C 180,E1 14960.33,E2 14960.33} C_VEL
LIN {X 0,Y 305.85,Z 565.696,A -85,B 0,C 180,E1 14962.076,E2 14962.076} C_VEL
LIN {X 0,Y 317.218,Z 582.047,A -85,B 0,C 180,E1 14967.058,E2 14967.058} C_VEL
LIN {X 0,Y 330.882,Z 602.857,A -85,B 0,C 180,E1 14971.941,E2 14971.941} C_VEL
LIN {X 0,Y 344.496,Z 629.045,A -85,B 0,C 180,E1 14976.649,E2 14976.649} C_VEL
LIN {X 0,Y 354.711,Z 657.933,A -85,B 0,C 180,E1 14980.847,E2 14980.847} C_VEL
LIN {X 0,Y 346.938,Z 695.058,A -85,B 0,C 180,E1 14983.489,E2 14983.489} C_VEL
LIN {X 0,Y 337.184,Z 729.985,A -85,B 0,C 180,E1 14987.013,E2 14987.013} C_VEL
LIN {X 0,Y 327.456,Z 760.138,A -85,B 0,C 180,E1 14991.26,E2 14991.26} C_VEL
LIN {X 0,Y 317.959,Z 787.837,A -85,B 0,C 180,E1 14996.64,E2 14996.64} C_VEL
LIN {X 0,Y 310.471,Z 810.699,A -85,B 0,C 180,E1 15002.795,E2 15002.795} C_VEL
LIN {X 0,Y 305.386,Z 828.917,A -85,B 0,C 180,E1 15009.694,E2 15009.694} C_VEL
LIN {X 0,Y 302.907,Z 841.289,A -85,B 0,C 180,E1 15016.655,E2 15016.655} C_VEL
LIN {X 0,Y 302.187,Z 847.922,A -85,B 0,C 180,E1 15022.805,E2 15022.805} C_VEL
LIN {X 0,Y 302.257,Z 850.659,A -85,B 0,C 180,E1 15030.001,E2 15030.001} C_VEL
LIN {X 0,Y 302.189,Z 847.93,A -85,B 0,C 180,E1 15037.196,E2 15037.196} C_VEL
LIN {X 0,Y 303.182,Z 839.727,A -85,B 0,C 180,E1 15044.46,E2 15044.46} C_VEL
LIN {X 0,Y 306.161,Z 825.682,A -85,B 0,C 180,E1 15051.771,E2 15051.771} C_VEL
LIN {X 0,Y 312.369,Z 804.847,A -85,B 0,C 180,E1 15058.993,E2 15058.993} C_VEL
LIN {X 0,Y 320.481,Z 780.623,A -85,B 0,C 180,E1 15064.948,E2 15064.948} C_VEL
LIN {X 0,Y 330.002,Z 752.495,A -85,B 0,C 180,E1 15069.966,E2 15069.966} C_VEL
LIN {X 0,Y 340.023,Z 720.486,A -85,B 0,C 180,E1 15074.088,E2 15074.088} C_VEL
LIN {X 0,Y 340.702,Z 718.33,A -85,B 0,C 180,E1 15074.314,E2 15074.314} C_VEL
LIN {X 0,Y 342.137,Z 707.928,A -85,B 0,C 180,E1 15075.627,E2 15075.627} C_VEL
LIN {X 0,Y 342.187,Z 692.263,A -85,B 0,C 180,E1 15077.666,E2 15077.666} C_VEL
LIN {X 0,Y 342.558,Z 690.341,A -85,B 0,C 180,E1 15077.833,E2 15077.833} C_VEL
LIN {X 0,Y 348.893,Z 661.305,A -85,B 0,C 180,E1 15079.875,E2 15079.875} C_VEL
LIN {X 0,Y 339.198,Z 632.895,A -85,B 0,C 180,E1 15084.208,E2 15084.208} C_VEL
LIN {X 0,Y 326.189,Z 606.993,A -85,B 0,C 180,E1 15089.097,E2 15089.097} C_VEL
LIN {X 0,Y 311.692,Z 584.38,A -85,B 0,C 180,E1 15094.752,E2 15094.752} C_VEL
LIN {X 0,Y 302.152,Z 571.138,A -85,B 0,C 180,E1 15099.275,E2 15099.275} C_VEL
LIN {X 0,Y 298.272,Z 565.366,A -85,B 0,C 180,E1 15101.504,E2 15101.504} C_VEL
LIN {X 0,Y 293.113,Z 559.566,A -85,B 0,C 180,E1 15104.832,E2 15104.832} C_VEL
LIN {X 0,Y 292.764,Z 557.03,A -85,B 0,C 180,E1 15105.398,E2 15105.398} C_VEL
LIN {X 0,Y 293.431,Z 557.03,A -85,B 0,C 180,E1 15114.077,E2 15114.077} C_VEL
LIN {X 0,Y 293.982,Z 557.03,A -85,B 0,C 180,E1 15119.999,E2 15119.999} C_VEL
LIN {X 0,Y 293.46,Z 557.03,A -85,B 0,C 180,E1 15125.922,E2 15125.922} C_VEL
LIN {X 0,Y 293.017,Z 557.03,A -85,B 0,C 180,E1 15131.927,E2 15131.927} C_VEL
LIN {X 0,Y 292.522,Z 557.088,A -85,B 0,C 180,E1 15138.97,E2 15138.97} C_VEL
LIN {X 0,Y 294.114,Z 561.819,A -85,B 0,C 180,E1 15140.331,E2 15140.331} C_VEL
LIN {X 0,Y 298.109,Z 565.468,A -85,B 0,C 180,E1 15142.782,E2 15142.782} C_VEL
LIN {X 0,Y 302.08,Z 571.247,A -85,B 0,C 180,E1 15145.04,E2 15145.04} C_VEL
LIN {X 0,Y 313.046,Z 586.344,A -85,B 0,C 180,E1 15150.115,E2 15150.115} C_VEL
LIN {X 0,Y 327.385,Z 609.088,A -85,B 0,C 180,E1 15155.719,E2 15155.719} C_VEL
LIN {X 0,Y 339.909,Z 635.259,A -85,B 0,C 180,E1 15160.689,E2 15160.689} C_VEL
LIN {X 0,Y 347.786,Z 659.472,A -85,B 0,C 180,E1 15164.581,E2 15164.581} C_VEL
LIN {X 0,Y 339.579,Z 692.883,A -85,B 0,C 180,E1 15167.357,E2 15167.357} C_VEL
LIN {X 0,Y 329.403,Z 723.982,A -85,B 0,C 180,E1 15171.013,E2 15171.013} C_VEL
LIN {X 0,Y 318.865,Z 751.801,A -85,B 0,C 180,E1 15175.713,E2 15175.713} C_VEL
LIN {X 0,Y 308.798,Z 776.043,A -85,B 0,C 180,E1 15181.647,E2 15181.647} C_VEL
LIN {X 0,Y 301.631,Z 793.749,A -85,B 0,C 180,E1 15187.986,E2 15187.986} C_VEL
LIN {X 0,Y 296.942,Z 807.029,A -85,B 0,C 180,E1 15195.229,E2 15195.229} C_VEL
LIN {X 0,Y 295.13,Z 813.578,A -85,B 0,C 180,E1 15201.146,E2 15201.146} C_VEL
LIN {X 0,Y 294.452,Z 816.757,A -85,B 0,C 180,E1 15207.052,E2 15207.052} C_VEL
LIN {X 0,Y 294.512,Z 816.718,A -85,B 0,C 180,E1 15212.946,E2 15212.946} C_VEL
LIN {X 0,Y 295.539,Z 812.148,A -85,B 0,C 180,E1 15220.329,E2 15220.329} C_VEL
LIN {X 0,Y 298.509,Z 802.197,A -85,B 0,C 180,E1 15227.717,E2 15227.717} C_VEL
LIN {X 0,Y 304.689,Z 786.054,A -85,B 0,C 180,E1 15234.984,E2 15234.984} C_VEL
LIN {X 0,Y 313.459,Z 764.785,A -85,B 0,C 180,E1 15241.281,E2 15241.281} C_VEL
LIN {X 0,Y 323.143,Z 740.663,A -85,B 0,C 180,E1 15246.265,E2 15246.265} C_VEL
LIN {X 0,Y 333.616,Z 711.576,A -85,B 0,C 180,E1 15250.507,E2 15250.507} C_VEL
LIN {X 0,Y 343.594,Z 677.995,A -85,B 0,C 180,E1 15253.9,E2 15253.9} C_VEL
LIN {X 0,Y 347.957,Z 660.325,A -85,B 0,C 180,E1 15255.179,E2 15255.179} C_VEL
LIN {X 0,Y 338.609,Z 632.144,A -85,B 0,C 180,E1 15259.735,E2 15259.735} C_VEL
LIN {X 0,Y 326.279,Z 607.242,A -85,B 0,C 180,E1 15264.55,E2 15264.55} C_VEL
LIN {X 0,Y 311.985,Z 584.715,A -85,B 0,C 180,E1 15270.173,E2 15270.173} C_VEL
LIN {X 0,Y 301.953,Z 571.152,A -85,B 0,C 180,E1 15274.844,E2 15274.844} C_VEL
LIN {X 0,Y 298.101,Z 565.558,A -85,B 0,C 180,E1 15277.02,E2 15277.02} C_VEL
LIN {X 0,Y 292.804,Z 559.118,A -85,B 0,C 180,E1 15280.46,E2 15280.46} C_VEL
LIN {X 0,Y 292.574,Z 557.03,A -85,B 0,C 180,E1 15281.131,E2 15281.131} C_VEL
LIN {X 0,Y 293.094,Z 557.03,A -85,B 0,C 180,E1 15288.957,E2 15288.957} C_VEL
LIN {X 0,Y 293.768,Z 557.03,A -85,B 0,C 180,E1 15297.046,E2 15297.046} C_VEL
LIN {X 0,Y 293.763,Z 557.03,A -85,B 0,C 180,E1 15302.955,E2 15302.955} C_VEL
LIN {X 0,Y 292.978,Z 557.03,A -85,B 0,C 180,E1 15311.929,E2 15311.929} C_VEL
LIN {X 0,Y 292.769,Z 557.266,A -85,B 0,C 180,E1 15314.889,E2 15314.889} C_VEL
LIN {X 0,Y 294.487,Z 562.025,A -85,B 0,C 180,E1 15316.312,E2 15316.312} C_VEL
LIN {X 0,Y 298.379,Z 565.794,A -85,B 0,C 180,E1 15318.681,E2 15318.681} C_VEL
LIN {X 0,Y 302.689,Z 571.501,A -85,B 0,C 180,E1 15321.07,E2 15321.07} C_VEL
LIN {X 0,Y 314.797,Z 589.166,A -85,B 0,C 180,E1 15326.607,E2 15326.607} C_VEL
LIN {X 0,Y 327.903,Z 610.253,A -85,B 0,C 180,E1 15331.603,E2 15331.603} C_VEL
LIN {X 0,Y 340.402,Z 635.791,A -85,B 0,C 180,E1 15336.306,E2 15336.306} C_VEL
LIN {X 0,Y 348.857,Z 661.259,A -85,B 0,C 180,E1 15340.137,E2 15340.137} C_VEL
LIN {X 0,Y 340.492,Z 697.807,A -85,B 0,C 180,E1 15342.803,E2 15342.803} C_VEL
LIN {X 0,Y 330.421,Z 732.048,A -85,B 0,C 180,E1 15346.38,E2 15346.38} C_VEL
LIN {X 0,Y 319.921,Z 762.868,A -85,B 0,C 180,E1 15350.898,E2 15350.898} C_VEL
LIN {X 0,Y 309.955,Z 790.661,A -85,B 0,C 180,E1 15356.59,E2 15356.59} C_VEL
LIN {X 0,Y 302.054,Z 813.573,A -85,B 0,C 180,E1 15363.185,E2 15363.185} C_VEL
LIN {X 0,Y 297.225,Z 830.587,A -85,B 0,C 180,E1 15370.159,E2 15370.159} C_VEL
LIN {X 0,Y 294.943,Z 842.119,A -85,B 0,C 180,E1 15377.234,E2 15377.234} C_VEL
LIN {X 0,Y 294.21,Z 848.405,A -85,B 0,C 180,E1 15384.093,E2 15384.093} C_VEL
LIN {X 0,Y 294.364,Z 850.216,A -85,B 0,C 180,E1 15390.001,E2 15390.001} C_VEL
LIN {X 0,Y 294.317,Z 847.484,A -85,B 0,C 180,E1 15397.39,E2 15397.39} C_VEL
LIN {X 0,Y 295.391,Z 839.269,A -85,B 0,C 180,E1 15404.85,E2 15404.85} C_VEL
LIN {X 0,Y 298.591,Z 825.207,A -85,B 0,C 180,E1 15412.353,E2 15412.353} C_VEL
LIN {X 0,Y 304.793,Z 805.604,A -85,B 0,C 180,E1 15419.377,E2 15419.377} C_VEL
LIN {X 0,Y 313.818,Z 780.099,A -85,B 0,C 180,E1 15425.803,E2 15425.803} C_VEL
LIN {X 0,Y 324.097,Z 750.907,A -85,B 0,C 180,E1 15431.055,E2 15431.055} C_VEL
LIN {X 0,Y 334.728,Z 718.512,A -85,B 0,C 180,E1 15435.189,E2 15435.189} C_VEL
LIN {X 0,Y 342.558,Z 690.341,A -85,B 0,C 180,E1 15437.833,E2 15437.833} C_VEL
LIN {X 0,Y 344.243,Z 675.079,A -85,B 0,C 180,E1 15439.302,E2 15439.302} C_VEL
LIN {X 0,Y 342.198,Z 661.211,A -85,B 0,C 180,E1 15441.116,E2 15441.116} C_VEL
LIN {X 0,Y 333.039,Z 634.655,A -85,B 0,C 180,E1 15445.432,E2 15445.432} C_VEL
LIN {X 0,Y 320.231,Z 608.838,A -85,B 0,C 180,E1 15450.643,E2 15450.643} C_VEL
LIN {X 0,Y 307.686,Z 589.486,A -85,B 0,C 180,E1 15455.953,E2 15455.953} C_VEL
LIN {X 0,Y 299.538,Z 577.924,A -85,B 0,C 180,E1 15460.052,E2 15460.052} C_VEL
LIN {X 0,Y 294.946,Z 571.418,A -85,B 0,C 180,E1 15462.833,E2 15462.833} C_VEL
LIN {X 0,Y 291.064,Z 566.12,A -85,B 0,C 180,E1 15465.599,E2 15465.599} C_VEL
LIN {X 0,Y 290.079,Z 564.447,A -85,B 0,C 180,E1 15466.416,E2 15466.416} C_VEL
LIN {X 0,Y 285.645,Z 559.68,A -85,B 0,C 180,E1 15470.532,E2 15470.532} C_VEL
LIN {X 0,Y 285.27,Z 557.03,A -85,B 0,C 180,E1 15471.607,E2 15471.607} C_VEL
LIN {X 0,Y 286.108,Z 557.03,A -85,B 0,C 180,E1 15479.999,E2 15479.999} C_VEL
LIN {X 0,Y 285.518,Z 557.03,A -85,B 0,C 180,E1 15486.087,E2 15486.087} C_VEL
LIN {X 0,Y 285.012,Z 557.709,A -85,B 0,C 180,E1 15492.949,E2 15492.949} C_VEL
LIN {X 0,Y 287.196,Z 562.672,A -85,B 0,C 180,E1 15495.582,E2 15495.582} C_VEL
LIN {X 0,Y 290.833,Z 565.803,A -85,B 0,C 180,E1 15498.577,E2 15498.577} C_VEL
LIN {X 0,Y 294.566,Z 571.297,A -85,B 0,C 180,E1 15501.283,E2 15501.283} C_VEL
LIN {X 0,Y 296.657,Z 574.114,A -85,B 0,C 180,E1 15502.603,E2 15502.603} C_VEL
LIN {X 0,Y 302.218,Z 581.862,A -85,B 0,C 180,E1 15505.71,E2 15505.71} C_VEL
LIN {X 0,Y 310.44,Z 593.343,A -85,B 0,C 180,E1 15509.588,E2 15509.588} C_VEL
LIN {X 0,Y 323.627,Z 615.22,A -85,B 0,C 180,E1 15515.153,E2 15515.153} C_VEL
LIN {X 0,Y 335.063,Z 640.468,A -85,B 0,C 180,E1 15520.117,E2 15520.117} C_VEL
LIN {X 0,Y 341.904,Z 663.654,A -85,B 0,C 180,E1 15523.945,E2 15523.945} C_VEL
LIN {X 0,Y 332.387,Z 698.191,A -85,B 0,C 180,E1 15526.9,E2 15526.9} C_VEL
LIN {X 0,Y 321.231,Z 730.003,A -85,B 0,C 180,E1 15530.939,E2 15530.939} C_VEL
LIN {X 0,Y 310.171,Z 757.173,A -85,B 0,C 180,E1 15535.932,E2 15535.932} C_VEL
LIN {X 0,Y 300.453,Z 779.569,A -85,B 0,C 180,E1 15541.871,E2 15541.871} C_VEL
LIN {X 0,Y 293.01,Z 797.248,A -85,B 0,C 180,E1 15548.794,E2 15548.794} C_VEL
LIN {X 0,Y 288.806,Z 808.803,A -85,B 0,C 180,E1 15555.811,E2 15555.811} C_VEL
LIN {X 0,Y 287.296,Z 814.023,A -85,B 0,C 180,E1 15560.903,E2 15560.903} C_VEL
LIN {X 0,Y 286.565,Z 817.2,A -85,B 0,C 180,E1 15566.971,E2 15566.971} C_VEL
LIN {X 0,Y 286.636,Z 817.161,A -85,B 0,C 180,E1 15573.027,E2 15573.027} C_VEL
LIN {X 0,Y 287.721,Z 812.597,A -85,B 0,C 180,E1 15580.613,E2 15580.613} C_VEL
LIN {X 0,Y 290.918,Z 802.653,A -85,B 0,C 180,E1 15588.195,E2 15588.195} C_VEL
LIN {X 0,Y 297.466,Z 786.524,A -85,B 0,C 180,E1 15595.634,E2 15595.634} C_VEL
LIN {X 0,Y 306.651,Z 765.279,A -85,B 0,C 180,E1 15602.057,E2 15602.057} C_VEL
LIN {X 0,Y 316.78,Z 741.186,A -85,B 0,C 180,E1 15607.114,E2 15607.114} C_VEL
LIN {X 0,Y 327.65,Z 712.16,A -85,B 0,C 180,E1 15611.404,E2 15611.404} C_VEL
LIN {X 0,Y 337.632,Z 679.92,A -85,B 0,C 180,E1 15614.715,E2 15614.715} C_VEL
LIN {X 0,Y 341.878,Z 663.603,A -85,B 0,C 180,E1 15615.947,E2 15615.947} C_VEL
LIN {X 0,Y 333.833,Z 637.439,A -85,B 0,C 180,E1 15620.317,E2 15620.317} C_VEL
LIN {X 0,Y 322.536,Z 613.328,A -85,B 0,C 180,E1 15625.157,E2 15625.157} C_VEL
LIN {X 0,Y 309.249,Z 591.436,A -85,B 0,C 180,E1 15630.79,E2 15630.79} C_VEL
LIN {X 0,Y 299.442,Z 578.01,A -85,B 0,C 180,E1 15635.586,E2 15635.586} C_VEL
LIN {X 0,Y 294.7,Z 571.385,A -85,B 0,C 180,E1 15638.431,E2 15638.431} C_VEL
LIN {X 0,Y 290.782,Z 565.695,A -85,B 0,C 180,E1 15641.228,E2 15641.228} C_VEL
LIN {X 0,Y 285.255,Z 559.127,A -85,B 0,C 180,E1 15646.281,E2 15646.281} C_VEL
LIN {X 0,Y 285.039,Z 557.03,A -85,B 0,C 180,E1 15646.955,E2 15646.955} C_VEL
LIN {X 0,Y 285.533,Z 557.03,A -85,B 0,C 180,E1 15653.913,E2 15653.913} C_VEL
LIN {X 0,Y 286.105,Z 557.03,A -85,B 0,C 180,E1 15660.001,E2 15660.001} C_VEL
LIN {X 0,Y 285.307,Z 557.03,A -85,B 0,C 180,E1 15668.776,E2 15668.776} C_VEL
LIN {X 0,Y 287.135,Z 562.337,A -85,B 0,C 180,E1 15671.305,E2 15671.305} C_VEL
LIN {X 0,Y 290.926,Z 565.604,A -85,B 0,C 180,E1 15674.408,E2 15674.408} C_VEL
LIN {X 0,Y 294.633,Z 571.196,A -85,B 0,C 180,E1 15677.089,E2 15677.089} C_VEL
LIN {X 0,Y 296.726,Z 573.974,A -85,B 0,C 180,E1 15678.403,E2 15678.403} C_VEL
LIN {X 0,Y 302.231,Z 581.77,A -85,B 0,C 180,E1 15681.488,E2 15681.488} C_VEL
LIN {X 0,Y 311.738,Z 595.451,A -85,B 0,C 180,E1 15685.918,E2 15685.918} C_VEL
LIN {X 0,Y 324.015,Z 615.959,A -85,B 0,C 180,E1 15690.929,E2 15690.929} C_VEL
LIN {X 0,Y 335.694,Z 641.134,A -85,B 0,C 180,E1 15695.725,E2 15695.725} C_VEL
LIN {X 0,Y 342.884,Z 663.828,A -85,B 0,C 180,E1 15699.296,E2 15699.296} C_VEL
LIN {X 0,Y 333.591,Z 702.289,A -85,B 0,C 180,E1 15702.238,E2 15702.238} C_VEL
LIN {X 0,Y 322.39,Z 737.905,A -85,B 0,C 180,E1 15706.219,E2 15706.219} C_VEL
LIN {X 0,Y 311.192,Z 768.708,A -85,B 0,C 180,E1 15711.115,E2 15711.115} C_VEL
LIN {X 0,Y 301.406,Z 794.625,A -85,B 0,C 180,E1 15716.888,E2 15716.888} C_VEL
LIN {X 0,Y 293.81,Z 815.76,A -85,B 0,C 180,E1 15723.451,E2 15723.451} C_VEL
LIN {X 0,Y 289.138,Z 831.713,A -85,B 0,C 180,E1 15730.476,E2 15730.476} C_VEL
LIN {X 0,Y 286.927,Z 842.726,A -85,B 0,C 180,E1 15737.815,E2 15737.815} C_VEL
LIN {X 0,Y 286.321,Z 847.958,A -85,B 0,C 180,E1 15743.93,E2 15743.93} C_VEL
LIN {X 0,Y 286.47,Z 849.773,A -85,B 0,C 180,E1 15750.001,E2 15750.001} C_VEL
LIN {X 0,Y 286.439,Z 847.037,A -85,B 0,C 180,E1 15757.594,E2 15757.594} C_VEL
LIN {X 0,Y 287.604,Z 838.812,A -85,B 0,C 180,E1 15765.262,E2 15765.262} C_VEL
LIN {X 0,Y 291.043,Z 824.731,A -85,B 0,C 180,E1 15772.965,E2 15772.965} C_VEL
LIN {X 0,Y 297.557,Z 805.225,A -85,B 0,C 180,E1 15780.123,E2 15780.123} C_VEL
LIN {X 0,Y 307.119,Z 779.75,A -85,B 0,C 180,E1 15786.663,E2 15786.663} C_VEL
LIN {X 0,Y 317.608,Z 751.36,A -85,B 0,C 180,E1 15791.866,E2 15791.866} C_VEL
LIN {X 0,Y 328.46,Z 719.649,A -85,B 0,C 180,E1 15796.004,E2 15796.004} C_VEL
LIN {X 0,Y 338.523,Z 684.397,A -85,B 0,C 180,E1 15799.248,E2 15799.248} C_VEL
LIN {X 0,Y 342.925,Z 664.012,A -85,B 0,C 180,E1 15800.703,E2 15800.703} C_VEL
LIN {X 0,Y 342.198,Z 661.211,A -85,B 0,C 180,E1 15801.116,E2 15801.116} C_VEL
LIN {X 0,Y 337.866,Z 653.452,A -85,B 0,C 180,E1 15802.747,E2 15802.747} C_VEL
LIN {X 0,Y 329.299,Z 642.085,A -85,B 0,C 180,E1 15805.669,E2 15805.669} C_VEL
LIN {X 0,Y 318.272,Z 618.132,A -85,B 0,C 180,E1 15810.568,E2 15810.568} C_VEL
LIN {X 0,Y 306.18,Z 597.704,A -85,B 0,C 180,E1 15816.021,E2 15816.021} C_VEL
LIN {X 0,Y 297.001,Z 584.528,A -85,B 0,C 180,E1 15820.843,E2 15820.843} C_VEL
LIN {X 0,Y 292.714,Z 578.464,A -85,B 0,C 180,E1 15823.569,E2 15823.569} C_VEL
LIN {X 0,Y 288.153,Z 571.924,A -85,B 0,C 180,E1 15827.097,E2 15827.097} C_VEL
LIN {X 0,Y 284.091,Z 566.738,A -85,B 0,C 180,E1 15831.186,E2 15831.186} C_VEL
LIN {X 0,Y 283.313,Z 564.675,A -85,B 0,C 180,E1 15832.322,E2 15832.322} C_VEL
LIN {X 0,Y 279.697,Z 561.653,A -85,B 0,C 180,E1 15839.999,E2 15839.999} C_VEL
LIN {X 0,Y 283.533,Z 565.148,A -85,B 0,C 180,E1 15852.332,E2 15852.332} C_VEL
LIN {X 0,Y 286.571,Z 570.991,A -85,B 0,C 180,E1 15855.918,E2 15855.918} C_VEL
LIN {X 0,Y 289.208,Z 573.451,A -85,B 0,C 180,E1 15858.123,E2 15858.123} C_VEL
LIN {X 0,Y 295.01,Z 581.868,A -85,B 0,C 180,E1 15862.258,E2 15862.258} C_VEL
LIN {X 0,Y 303.692,Z 593.872,A -85,B 0,C 180,E1 15867.057,E2 15867.057} C_VEL
LIN {X 0,Y 315.731,Z 613.785,A -85,B 0,C 180,E1 15872.747,E2 15872.747} C_VEL
LIN {X 0,Y 326.241,Z 635.473,A -85,B 0,C 180,E1 15877.564,E2 15877.564} C_VEL
LIN {X 0,Y 334.849,Z 661.139,A -85,B 0,C 180,E1 15882.263,E2 15882.263} C_VEL
LIN {X 0,Y 335.757,Z 667.523,A -85,B 0,C 180,E1 15883.196,E2 15883.196} C_VEL
LIN {X 0,Y 325.555,Z 702.029,A -85,B 0,C 180,E1 15886.307,E2 15886.307} C_VEL
LIN {X 0,Y 314.326,Z 732.449,A -85,B 0,C 180,E1 15890.329,E2 15890.329} C_VEL
LIN {X 0,Y 302.979,Z 759.074,A -85,B 0,C 180,E1 15895.403,E2 15895.403} C_VEL
LIN {X 0,Y 292.627,Z 781.875,A -85,B 0,C 180,E1 15901.747,E2 15901.747} C_VEL
LIN {X 0,Y 284.933,Z 799.162,A -85,B 0,C 180,E1 15908.98,E2 15908.98} C_VEL
LIN {X 0,Y 280.846,Z 809.937,A -85,B 0,C 180,E1 15916.003,E2 15916.003} C_VEL
LIN {X 0,Y 278.959,Z 816.445,A -85,B 0,C 180,E1 15923.768,E2 15923.768} C_VEL
LIN {X 0,Y 278.731,Z 818.055,A -85,B 0,C 180,E1 15929.999,E2 15929.999} C_VEL
LIN {X 0,Y 279.247,Z 815.514,A -85,B 0,C 180,E1 15937.79,E2 15937.79} C_VEL
LIN {X 0,Y 281.602,Z 807.783,A -85,B 0,C 180,E1 15945.594,E2 15945.594} C_VEL
LIN {X 0,Y 286.188,Z 796.086,A -85,B 0,C 180,E1 15952.454,E2 15952.454} C_VEL
LIN {X 0,Y 293.663,Z 779.465,A -85,B 0,C 180,E1 15958.936,E2 15958.936} C_VEL
LIN {X 0,Y 303.324,Z 758.131,A -85,B 0,C 180,E1 15964.702,E2 15964.702} C_VEL
LIN {X 0,Y 314.242,Z 732.431,A -85,B 0,C 180,E1 15969.571,E2 15969.571} C_VEL
LIN {X 0,Y 325.406,Z 702.231,A -85,B 0,C 180,E1 15973.566,E2 15973.566} C_VEL
LIN {X 0,Y 335.188,Z 669.366,A -85,B 0,C 180,E1 15976.556,E2 15976.556} C_VEL
LIN {X 0,Y 335.469,Z 663.808,A -85,B 0,C 180,E1 15977.176,E2 15977.176} C_VEL
LIN {X 0,Y 327.037,Z 637.461,A -85,B 0,C 180,E1 15981.908,E2 15981.908} C_VEL
LIN {X 0,Y 316.021,Z 614.235,A -85,B 0,C 180,E1 15986.98,E2 15986.98} C_VEL
LIN {X 0,Y 302.925,Z 592.536,A -85,B 0,C 180,E1 15993.17,E2 15993.17} C_VEL
LIN {X 0,Y 292.731,Z 578.64,A -85,B 0,C 180,E1 15999.019,E2 15999.019} C_VEL
LIN {X 0,Y 288.078,Z 571.922,A -85,B 0,C 180,E1 16002.572,E2 16002.572} C_VEL
LIN {X 0,Y 283.829,Z 566.498,A -85,B 0,C 180,E1 16006.8,E2 16006.8} C_VEL
LIN {X 0,Y 283.26,Z 564.693,A -85,B 0,C 180,E1 16007.656,E2 16007.656} C_VEL
LIN {X 0,Y 279.466,Z 561.32,A -85,B 0,C 180,E1 16020.001,E2 16020.001} C_VEL
LIN {X 0,Y 283.827,Z 565.596,A -85,B 0,C 180,E1 16028.629,E2 16028.629} C_VEL
LIN {X 0,Y 286.864,Z 571.016,A -85,B 0,C 180,E1 16031.994,E2 16031.994} C_VEL
LIN {X 0,Y 289.303,Z 573.405,A -85,B 0,C 180,E1 16034.007,E2 16034.007} C_VEL
LIN {X 0,Y 293.819,Z 579.253,A -85,B 0,C 180,E1 16037.235,E2 16037.235} C_VEL
LIN {X 0,Y 304.654,Z 595.646,A -85,B 0,C 180,E1 16043.329,E2 16043.329} C_VEL
LIN {X 0,Y 316.616,Z 614.935,A -85,B 0,C 180,E1 16048.752,E2 16048.752} C_VEL
LIN {X 0,Y 328.461,Z 640.176,A -85,B 0,C 180,E1 16054.003,E2 16054.003} C_VEL
LIN {X 0,Y 336.853,Z 666.167,A -85,B 0,C 180,E1 16058.374,E2 16058.374} C_VEL
LIN {X 0,Y 334.672,Z 678.069,A -85,B 0,C 180,E1 16059.296,E2 16059.296} C_VEL
LIN {X 0,Y 323.971,Z 715.266,A -85,B 0,C 180,E1 16062.544,E2 16062.544} C_VEL
LIN {X 0,Y 312.046,Z 749.373,A -85,B 0,C 180,E1 16066.922,E2 16066.922} C_VEL
LIN {X 0,Y 300.98,Z 777.899,A -85,B 0,C 180,E1 16072.119,E2 16072.119} C_VEL
LIN {X 0,Y 291.454,Z 802.049,A -85,B 0,C 180,E1 16078.267,E2 16078.267} C_VEL
LIN {X 0,Y 284.685,Z 820.566,A -85,B 0,C 180,E1 16084.82,E2 16084.82} C_VEL
LIN {X 0,Y 280.603,Z 834.727,A -85,B 0,C 180,E1 16091.926,E2 16091.926} C_VEL
LIN {X 0,Y 278.842,Z 844,A -85,B 0,C 180,E1 16099.094,E2 16099.094} C_VEL
LIN {X 0,Y 278.432,Z 847.511,A -85,B 0,C 180,E1 16103.757,E2 16103.757} C_VEL
LIN {X 0,Y 278.577,Z 849.33,A -85,B 0,C 180,E1 16110.001,E2 16110.001} C_VEL
LIN {X 0,Y 278.546,Z 846.59,A -85,B 0,C 180,E1 16117.811,E2 16117.811} C_VEL
LIN {X 0,Y 279.839,Z 838.355,A -85,B 0,C 180,E1 16125.696,E2 16125.696} C_VEL
LIN {X 0,Y 283.506,Z 824.255,A -85,B 0,C 180,E1 16133.612,E2 16133.612} C_VEL
LIN {X 0,Y 290.51,Z 804.732,A -85,B 0,C 180,E1 16140.932,E2 16140.932} C_VEL
LIN {X 0,Y 300.451,Z 779.359,A -85,B 0,C 180,E1 16147.578,E2 16147.578} C_VEL
LIN {X 0,Y 311.521,Z 750.794,A -85,B 0,C 180,E1 16152.878,E2 16152.878} C_VEL
LIN {X 0,Y 323.028,Z 718.602,A -85,B 0,C 180,E1 16157.084,E2 16157.084} C_VEL
LIN {X 0,Y 333.343,Z 683.652,A -85,B 0,C 180,E1 16160.292,E2 16160.292} C_VEL
LIN {X 0,Y 337.187,Z 667.363,A -85,B 0,C 180,E1 16161.465,E2 16161.465} C_VEL
LIN {X 0,Y 329.299,Z 642.085,A -85,B 0,C 180,E1 16165.669,E2 16165.669} C_VEL
LIN {X 0,Y 324.35,Z 635.559,A -85,B 0,C 180,E1 16167.472,E2 16167.472} C_VEL
LIN {X 0,Y 316.184,Z 627.528,A -85,B 0,C 180,E1 16170.393,E2 16170.393} C_VEL
LIN {X 0,Y 315.532,Z 626.221,A -85,B 0,C 180,E1 16170.694,E2 16170.694} C_VEL
LIN {X 0,Y 303.719,Z 604.743,A -85,B 0,C 180,E1 16176.498,E2 16176.498} C_VEL
LIN {X 0,Y 294.521,Z 591.089,A -85,B 0,C 180,E1 16181.648,E2 16181.648} C_VEL
LIN {X 0,Y 290.799,Z 585.716,A -85,B 0,C 180,E1 16184.137,E2 16184.137} C_VEL
LIN {X 0,Y 286.511,Z 579.443,A -85,B 0,C 180,E1 16187.604,E2 16187.604} C_VEL
LIN {X 0,Y 282.562,Z 573.68,A -85,B 0,C 180,E1 16191.883,E2 16191.883} C_VEL
LIN {X 0,Y 281.212,Z 572.033,A -85,B 0,C 180,E1 16193.818,E2 16193.818} C_VEL
LIN {X 0,Y 278.731,Z 569.523,A -85,B 0,C 180,E1 16199.999,E2 16199.999} C_VEL
LIN {X 0,Y 282.203,Z 572.765,A -85,B 0,C 180,E1 16211.873,E2 16211.873} C_VEL
LIN {X 0,Y 285.491,Z 578.81,A -85,B 0,C 180,E1 16215.829,E2 16215.829} C_VEL
LIN {X 0,Y 287.813,Z 581.445,A -85,B 0,C 180,E1 16217.847,E2 16217.847} C_VEL
LIN {X 0,Y 293.19,Z 589.27,A -85,B 0,C 180,E1 16221.805,E2 16221.805} C_VEL
LIN {X 0,Y 301.463,Z 601.396,A -85,B 0,C 180,E1 16226.669,E2 16226.669} C_VEL
LIN {X 0,Y 312.111,Z 619.982,A -85,B 0,C 180,E1 16232.144,E2 16232.144} C_VEL
LIN {X 0,Y 322.018,Z 641.895,A -85,B 0,C 180,E1 16237.16,E2 16237.16} C_VEL
